LIN {X 0,Y 215.82,Z 913.097,A -85,B 0,C 180,E1 -20872.515,E2 -20872.515} C_VEL
LIN {X 0,Y 216.732,Z 913.858,A -85,B 0,C 180,E1 -20874.417,E2 -20874.417} C_VEL
LIN {X 0,Y 218.187,Z 914.153,A -85,B 0,C 180,E1 -20876.945,E2 -20876.945} C_VEL
LIN {X 0,Y 220.423,Z 913.484,A -85,B 0,C 180,E1 -20880,E2 -20880} C_VEL
LIN {X 0,Y 223.697,Z 911.017,A -85,B 0,C 180,E1 -20883.602,E2 -20883.602} C_VEL
LIN {X 0,Y 226.039,Z 908.76,A -85,B 0,C 180,E1 -20885.743,E2 -20885.743} C_VEL
LIN {X 0,Y 228.842,Z 905.544,A -85,B 0,C 180,E1 -20887.943,E2 -20887.943} C_VEL
LIN {X 0,Y 232.45,Z 900.63,A -85,B 0,C 180,E1 -20890.451,E2 -20890.451} C_VEL
LIN {X 0,Y 236.309,Z 894.485,A -85,B 0,C 180,E1 -20892.888,E2 -20892.888} C_VEL
LIN {X 0,Y 240.084,Z 887.75,A -85,B 0,C 180,E1 -20894.973,E2 -20894.973} C_VEL
LIN {X 0,Y 243.557,Z 880.667,A -85,B 0,C 180,E1 -20896.771,E2 -20896.771} C_VEL
LIN {X 0,Y 246.66,Z 873.613,A -85,B 0,C 180,E1 -20898.265,E2 -20898.265} C_VEL
LIN {X 0,Y 249.838,Z 865.279,A -85,B 0,C 180,E1 -20899.728,E2 -20899.728} C_VEL
LIN {X 0,Y 252.697,Z 856.675,A -85,B 0,C 180,E1 -20900.982,E2 -20900.982} C_VEL
LIN {X 0,Y 255.577,Z 846.343,A -85,B 0,C 180,E1 -20902.216,E2 -20902.216} C_VEL
LIN {X 0,Y 257.749,Z 836.491,A -85,B 0,C 180,E1 -20903.183,E2 -20903.183} C_VEL
LIN {X 0,Y 258.881,Z 830.775,A -85,B 0,C 180,E1 -20903.651,E2 -20903.651} C_VEL
LIN {X 0,Y 259.433,Z 825.363,A -85,B 0,C 180,E1 -20904.174,E2 -20904.174} C_VEL
LIN {X 0,Y 259.323,Z 808.224,A -85,B 0,C 180,E1 -20906.374,E2 -20906.374} C_VEL
LIN {X 0,Y 259.902,Z 802.661,A -85,B 0,C 180,E1 -20906.763,E2 -20906.763} C_VEL
LIN {X 0,Y 261.287,Z 793.546,A -85,B 0,C 180,E1 -20907.21,E2 -20907.21} C_VEL
LIN {X 0,Y 259.496,Z 789.462,A -85,B 0,C 180,E1 -20909.048,E2 -20909.048} C_VEL
LIN {X 0,Y 258.611,Z 787.722,A -85,B 0,C 180,E1 -20910.062,E2 -20910.062} C_VEL
LIN {X 0,Y 257.462,Z 785.023,A -85,B 0,C 180,E1 -20911.841,E2 -20911.841} C_VEL
LIN {X 0,Y 256.142,Z 782.443,A -85,B 0,C 180,E1 -20915.183,E2 -20915.183} C_VEL
LIN {X 0,Y 255.755,Z 782.963,A -85,B 0,C 180,E1 -20917.889,E2 -20917.889} C_VEL
LIN {X 0,Y 256.35,Z 784.832,A -85,B 0,C 180,E1 -20920.768,E2 -20920.768} C_VEL
LIN {X 0,Y 257.554,Z 788.257,A -85,B 0,C 180,E1 -20923.294,E2 -20923.294} C_VEL
LIN {X 0,Y 258.154,Z 798.129,A -85,B 0,C 180,E1 -20925.703,E2 -20925.703} C_VEL
LIN {X 0,Y 256.979,Z 813.634,A -85,B 0,C 180,E1 -20927.292,E2 -20927.292} C_VEL
LIN {X 0,Y 255.567,Z 830.787,A -85,B 0,C 180,E1 -20928.783,E2 -20928.783} C_VEL
LIN {X 0,Y 253.729,Z 848.64,A -85,B 0,C 180,E1 -20929.988,E2 -20929.988} C_VEL
LIN {X 0,Y 251.045,Z 862.414,A -85,B 0,C 180,E1 -20930.697,E2 -20930.697} C_VEL
LIN {X 0,Y 247.953,Z 874.211,A -85,B 0,C 180,E1 -20931.42,E2 -20931.42} C_VEL
LIN {X 0,Y 244.407,Z 885.491,A -85,B 0,C 180,E1 -20932.332,E2 -20932.332} C_VEL
LIN {X 0,Y 240.95,Z 894.919,A -85,B 0,C 180,E1 -20933.275,E2 -20933.275} C_VEL
LIN {X 0,Y 236.566,Z 905.538,A -85,B 0,C 180,E1 -20934.595,E2 -20934.595} C_VEL
LIN {X 0,Y 232.488,Z 914.575,A -85,B 0,C 180,E1 -20935.993,E2 -20935.993} C_VEL
LIN {X 0,Y 228.672,Z 922.392,A -85,B 0,C 180,E1 -20937.46,E2 -20937.46} C_VEL
LIN {X 0,Y 224.196,Z 930.838,A -85,B 0,C 180,E1 -20939.373,E2 -20939.373} C_VEL
LIN {X 0,Y 220.295,Z 938.075,A -85,B 0,C 180,E1 -20941.407,E2 -20941.407} C_VEL
LIN {X 0,Y 216.754,Z 944.309,A -85,B 0,C 180,E1 -20943.521,E2 -20943.521} C_VEL
LIN {X 0,Y 213.717,Z 949.729,A -85,B 0,C 180,E1 -20945.726,E2 -20945.726} C_VEL
LIN {X 0,Y 210.73,Z 955.112,A -85,B 0,C 180,E1 -20948.475,E2 -20948.475} C_VEL
LIN {X 0,Y 208.341,Z 959.496,A -85,B 0,C 180,E1 -20951.306,E2 -20951.306} C_VEL
LIN {X 0,Y 206.818,Z 962.938,A -85,B 0,C 180,E1 -20954.223,E2 -20954.223} C_VEL
LIN {X 0,Y 205.688,Z 966.163,A -85,B 0,C 180,E1 -20958.167,E2 -20958.167} C_VEL
LIN {X 0,Y 205.748,Z 967.832,A -85,B 0,C 180,E1 -20961.564,E2 -20961.564} C_VEL
LIN {X 0,Y 205.939,Z 970.43,A -85,B 0,C 180,E1 -20964.121,E2 -20964.121} C_VEL
LIN {X 0,Y 206.207,Z 971.913,A -85,B 0,C 180,E1 -20966.089,E2 -20966.089} C_VEL
LIN {X 0,Y 206.454,Z 972.92,A -85,B 0,C 180,E1 -20968.046,E2 -20968.046} C_VEL
LIN {X 0,Y 206.718,Z 973.5,A -85,B 0,C 180,E1 -20969.997,E2 -20969.997} C_VEL
LIN {X 0,Y 206.4,Z 973.571,A -85,B 0,C 180,E1 -20971.948,E2 -20971.948} C_VEL
LIN {X 0,Y 206.129,Z 973.197,A -85,B 0,C 180,E1 -20973.907,E2 -20973.907} C_VEL
LIN {X 0,Y 205.527,Z 971.148,A -85,B 0,C 180,E1 -20977.859,E2 -20977.859} C_VEL
LIN {X 0,Y 205.533,Z 968.537,A -85,B 0,C 180,E1 -20980.837,E2 -20980.837} C_VEL
LIN {X 0,Y 206.046,Z 964.96,A -85,B 0,C 180,E1 -20983.81,E2 -20983.81} C_VEL
LIN {X 0,Y 207.188,Z 960.35,A -85,B 0,C 180,E1 -20986.755,E2 -20986.755} C_VEL
LIN {X 0,Y 208.926,Z 954.588,A -85,B 0,C 180,E1 -20989.654,E2 -20989.654} C_VEL
LIN {X 0,Y 211.427,Z 947.534,A -85,B 0,C 180,E1 -20992.471,E2 -20992.471} C_VEL
LIN {X 0,Y 214.497,Z 938.894,A -85,B 0,C 180,E1 -20995.207,E2 -20995.207} C_VEL
LIN {X 0,Y 217.552,Z 930.1,A -85,B 0,C 180,E1 -20997.406,E2 -20997.406} C_VEL
LIN {X 0,Y 221.071,Z 919.363,A -85,B 0,C 180,E1 -20999.518,E2 -20999.518} C_VEL
LIN {X 0,Y 224.586,Z 907.346,A -85,B 0,C 180,E1 -21001.345,E2 -21001.345} C_VEL
LIN {X 0,Y 227.546,Z 895.307,A -85,B 0,C 180,E1 -21002.715,E2 -21002.715} C_VEL
LIN {X 0,Y 229.807,Z 883.048,A -85,B 0,C 180,E1 -21003.778,E2 -21003.778} C_VEL
LIN {X 0,Y 231.633,Z 869.859,A -85,B 0,C 180,E1 -21004.57,E2 -21004.57} C_VEL
LIN {X 0,Y 232.714,Z 855.087,A -85,B 0,C 180,E1 -21005.118,E2 -21005.118} C_VEL
LIN {X 0,Y 233.372,Z 840.252,A -85,B 0,C 180,E1 -21005.6,E2 -21005.6} C_VEL
LIN {X 0,Y 232.16,Z 817.156,A -85,B 0,C 180,E1 -21006.833,E2 -21006.833} C_VEL
LIN {X 0,Y 230.572,Z 796.33,A -85,B 0,C 180,E1 -21008.093,E2 -21008.093} C_VEL
LIN {X 0,Y 228.613,Z 780.544,A -85,B 0,C 180,E1 -21009.258,E2 -21009.258} C_VEL
LIN {X 0,Y 224.716,Z 771.185,A -85,B 0,C 180,E1 -21010.671,E2 -21010.671} C_VEL
LIN {X 0,Y 220.27,Z 761.8,A -85,B 0,C 180,E1 -21012.341,E2 -21012.341} C_VEL
LIN {X 0,Y 216.362,Z 754.458,A -85,B 0,C 180,E1 -21013.9,E2 -21013.9} C_VEL
LIN {X 0,Y 213.79,Z 749.36,A -85,B 0,C 180,E1 -21015.11,E2 -21015.11} C_VEL
LIN {X 0,Y 211.962,Z 742.772,A -85,B 0,C 180,E1 -21018.461,E2 -21018.461} C_VEL
LIN {X 0,Y 209.608,Z 735.268,A -85,B 0,C 180,E1 -21022.877,E2 -21022.877} C_VEL
LIN {X 0,Y 207.43,Z 729.065,A -85,B 0,C 180,E1 -21027.173,E2 -21027.173} C_VEL
LIN {X 0,Y 206.745,Z 726.767,A -85,B 0,C 180,E1 -21029.101,E2 -21029.101} C_VEL
LIN {X 0,Y 206.723,Z 726.734,A -85,B 0,C 180,E1 -21033.771,E2 -21033.771} C_VEL
LIN {X 0,Y 206.747,Z 726.723,A -85,B 0,C 180,E1 -21038.042,E2 -21038.042} C_VEL
LIN {X 0,Y 206.866,Z 726.706,A -85,B 0,C 180,E1 -21042.196,E2 -21042.196} C_VEL
LIN {X 0,Y 206.885,Z 726.703,A -85,B 0,C 180,E1 -21046.244,E2 -21046.244} C_VEL
LIN {X 0,Y 207.088,Z 726.677,A -85,B 0,C 180,E1 -21050.231,E2 -21050.231} C_VEL
LIN {X 0,Y 207.055,Z 726.689,A -85,B 0,C 180,E1 -21054.156,E2 -21054.156} C_VEL
LIN {X 0,Y 207.371,Z 726.655,A -85,B 0,C 180,E1 -21058.058,E2 -21058.058} C_VEL
LIN {X 0,Y 207.504,Z 726.623,A -85,B 0,C 180,E1 -21060,E2 -21060} C_VEL
LIN {X 0,Y 207.371,Z 726.65,A -85,B 0,C 180,E1 -21061.943,E2 -21061.943} C_VEL
LIN {X 0,Y 207.157,Z 726.672,A -85,B 0,C 180,E1 -21067.8,E2 -21067.8} C_VEL
LIN {X 0,Y 206.933,Z 726.7,A -85,B 0,C 180,E1 -21071.758,E2 -21071.758} C_VEL
LIN {X 0,Y 206.906,Z 726.717,A -85,B 0,C 180,E1 -21077.291,E2 -21077.291} C_VEL
LIN {X 0,Y 206.927,Z 727.223,A -85,B 0,C 180,E1 -21078.182,E2 -21078.182} C_VEL
LIN {X 0,Y 207.868,Z 729.668,A -85,B 0,C 180,E1 -21078.896,E2 -21078.896} C_VEL
LIN {X 0,Y 209.947,Z 731.814,A -85,B 0,C 180,E1 -21079.812,E2 -21079.812} C_VEL
LIN {X 0,Y 210.664,Z 732.614,A -85,B 0,C 180,E1 -21080.123,E2 -21080.123} C_VEL
LIN {X 0,Y 212.757,Z 735.862,A -85,B 0,C 180,E1 -21081.054,E2 -21081.054} C_VEL
LIN {X 0,Y 214.374,Z 737.753,A -85,B 0,C 180,E1 -21081.704,E2 -21081.704} C_VEL
LIN {X 0,Y 218.102,Z 743.058,A -85,B 0,C 180,E1 -21083.187,E2 -21083.187} C_VEL
LIN {X 0,Y 221.441,Z 747.9,A -85,B 0,C 180,E1 -21084.428,E2 -21084.428} C_VEL
LIN {X 0,Y 227.298,Z 757.078,A -85,B 0,C 180,E1 -21086.467,E2 -21086.467} C_VEL
LIN {X 0,Y 234.437,Z 769.956,A -85,B 0,C 180,E1 -21088.764,E2 -21088.764} C_VEL
LIN {X 0,Y 236.607,Z 774.439,A -85,B 0,C 180,E1 -21089.441,E2 -21089.441} C_VEL
LIN {X 0,Y 235.209,Z 812.585,A -85,B 0,C 180,E1 -21090.792,E2 -21090.792} C_VEL
LIN {X 0,Y 234.483,Z 825.574,A -85,B 0,C 180,E1 -21091.539,E2 -21091.539} C_VEL
LIN {X 0,Y 233.062,Z 838.159,A -85,B 0,C 180,E1 -21092.588,E2 -21092.588} C_VEL
LIN {X 0,Y 231.265,Z 849.427,A -85,B 0,C 180,E1 -21093.845,E2 -21093.845} C_VEL
LIN {X 0,Y 229.188,Z 859.482,A -85,B 0,C 180,E1 -21095.269,E2 -21095.269} C_VEL
LIN {X 0,Y 226.691,Z 869.468,A -85,B 0,C 180,E1 -21097.035,E2 -21097.035} C_VEL
LIN {X 0,Y 223.982,Z 878.589,A -85,B 0,C 180,E1 -21099.054,E2 -21099.054} C_VEL
LIN {X 0,Y 221.064,Z 887.18,A -85,B 0,C 180,E1 -21101.439,E2 -21101.439} C_VEL
LIN {X 0,Y 218.03,Z 895.011,A -85,B 0,C 180,E1 -21104.18,E2 -21104.18} C_VEL
LIN {X 0,Y 215.643,Z 900.847,A -85,B 0,C 180,E1 -21106.815,E2 -21106.815} C_VEL
LIN {X 0,Y 213.002,Z 906.39,A -85,B 0,C 180,E1 -21110.087,E2 -21110.087} C_VEL
LIN {X 0,Y 211.04,Z 910.178,A -85,B 0,C 180,E1 -21113.175,E2 -21113.175} C_VEL
LIN {X 0,Y 209.998,Z 912.106,A -85,B 0,C 180,E1 -21115.328,E2 -21115.328} C_VEL
LIN {X 0,Y 209.141,Z 913.446,A -85,B 0,C 180,E1 -21117.479,E2 -21117.479} C_VEL
LIN {X 0,Y 208.448,Z 914.316,A -85,B 0,C 180,E1 -21119.623,E2 -21119.623} C_VEL
LIN {X 0,Y 207.976,Z 914.685,A -85,B 0,C 180,E1 -21121.768,E2 -21121.768} C_VEL
LIN {X 0,Y 207.701,Z 914.563,A -85,B 0,C 180,E1 -21123.907,E2 -21123.907} C_VEL
LIN {X 0,Y 207.586,Z 913.993,A -85,B 0,C 180,E1 -21126.081,E2 -21126.081} C_VEL
LIN {X 0,Y 207.696,Z 912.944,A -85,B 0,C 180,E1 -21128.151,E2 -21128.151} C_VEL
LIN {X 0,Y 208.071,Z 910.751,A -85,B 0,C 180,E1 -21131.043,E2 -21131.043} C_VEL
LIN {X 0,Y 209.058,Z 906.954,A -85,B 0,C 180,E1 -21134.402,E2 -21134.402} C_VEL
LIN {X 0,Y 210.273,Z 902.255,A -85,B 0,C 180,E1 -21137.455,E2 -21137.455} C_VEL
LIN {X 0,Y 211.895,Z 896.255,A -85,B 0,C 180,E1 -21140.457,E2 -21140.457} C_VEL
LIN {X 0,Y 213.803,Z 888.74,A -85,B 0,C 180,E1 -21143.396,E2 -21143.396} C_VEL
LIN {X 0,Y 216.063,Z 879.378,A -85,B 0,C 180,E1 -21146.273,E2 -21146.273} C_VEL
LIN {X 0,Y 218.269,Z 869.484,A -85,B 0,C 180,E1 -21148.663,E2 -21148.663} C_VEL
LIN {X 0,Y 220.257,Z 858.973,A -85,B 0,C 180,E1 -21150.688,E2 -21150.688} C_VEL
LIN {X 0,Y 222.265,Z 847.005,A -85,B 0,C 180,E1 -21152.495,E2 -21152.495} C_VEL
LIN {X 0,Y 223.878,Z 834.316,A -85,B 0,C 180,E1 -21153.94,E2 -21153.94} C_VEL
LIN {X 0,Y 224.921,Z 821.294,A -85,B 0,C 180,E1 -21155.044,E2 -21155.044} C_VEL
LIN {X 0,Y 225.492,Z 807.746,A -85,B 0,C 180,E1 -21155.793,E2 -21155.793} C_VEL
LIN {X 0,Y 226.498,Z 770.265,A -85,B 0,C 180,E1 -21157.076,E2 -21157.076} C_VEL
LIN {X 0,Y 226.553,Z 765.8,A -85,B 0,C 180,E1 -21157.236,E2 -21157.236} C_VEL
LIN {X 0,Y 222.198,Z 756.35,A -85,B 0,C 180,E1 -21158.222,E2 -21158.222} C_VEL
LIN {X 0,Y 213.824,Z 739.599,A -85,B 0,C 180,E1 -21160.191,E2 -21160.191} C_VEL
LIN {X 0,Y 208.363,Z 730.146,A -85,B 0,C 180,E1 -21161.514,E2 -21161.514} C_VEL
LIN {X 0,Y 207.034,Z 727.418,A -85,B 0,C 180,E1 -21161.941,E2 -21161.941} C_VEL
LIN {X 0,Y 206.907,Z 726.757,A -85,B 0,C 180,E1 -21162.384,E2 -21162.384} C_VEL
LIN {X 0,Y 206.814,Z 726.719,A -85,B 0,C 180,E1 -21167.915,E2 -21167.915} C_VEL
LIN {X 0,Y 206.732,Z 726.734,A -85,B 0,C 180,E1 -21173.38,E2 -21173.38} C_VEL
LIN {X 0,Y 206.685,Z 726.721,A -85,B 0,C 180,E1 -21178.431,E2 -21178.431} C_VEL
LIN {X 0,Y 206.699,Z 726.709,A -85,B 0,C 180,E1 -21182.961,E2 -21182.961} C_VEL
LIN {X 0,Y 206.707,Z 726.693,A -85,B 0,C 180,E1 -21185.313,E2 -21185.313} C_VEL
LIN {X 0,Y 206.654,Z 726.743,A -85,B 0,C 180,E1 -21190.256,E2 -21190.256} C_VEL
LIN {X 0,Y 206.637,Z 726.746,A -85,B 0,C 180,E1 -21194.418,E2 -21194.418} C_VEL
LIN {X 0,Y 206.706,Z 726.866,A -85,B 0,C 180,E1 -21197.499,E2 -21197.499} C_VEL
LIN {X 0,Y 206.93,Z 727.899,A -85,B 0,C 180,E1 -21197.85,E2 -21197.85} C_VEL
LIN {X 0,Y 216.887,Z 756.802,A -85,B 0,C 180,E1 -21200.104,E2 -21200.104} C_VEL
LIN {X 0,Y 214.902,Z 807.381,A -85,B 0,C 180,E1 -21202.586,E2 -21202.586} C_VEL
LIN {X 0,Y 214.443,Z 818.809,A -85,B 0,C 180,E1 -21203.411,E2 -21203.411} C_VEL
LIN {X 0,Y 213.661,Z 829.523,A -85,B 0,C 180,E1 -21204.421,E2 -21204.421} C_VEL
LIN {X 0,Y 212.813,Z 839.899,A -85,B 0,C 180,E1 -21205.655,E2 -21205.655} C_VEL
LIN {X 0,Y 211.854,Z 849.82,A -85,B 0,C 180,E1 -21207.096,E2 -21207.096} C_VEL
LIN {X 0,Y 210.982,Z 858.654,A -85,B 0,C 180,E1 -21208.635,E2 -21208.635} C_VEL
LIN {X 0,Y 210.053,Z 867.479,A -85,B 0,C 180,E1 -21210.454,E2 -21210.454} C_VEL
LIN {X 0,Y 209.101,Z 875.776,A -85,B 0,C 180,E1 -21212.474,E2 -21212.474} C_VEL
LIN {X 0,Y 208.331,Z 882.894,A -85,B 0,C 180,E1 -21214.521,E2 -21214.521} C_VEL
LIN {X 0,Y 207.784,Z 889.046,A -85,B 0,C 180,E1 -21216.582,E2 -21216.582} C_VEL
LIN {X 0,Y 207.253,Z 895.478,A -85,B 0,C 180,E1 -21219.141,E2 -21219.141} C_VEL
LIN {X 0,Y 206.951,Z 901.32,A -85,B 0,C 180,E1 -21221.973,E2 -21221.973} C_VEL
LIN {X 0,Y 206.941,Z 905.217,A -85,B 0,C 180,E1 -21224.235,E2 -21224.235} C_VEL
LIN {X 0,Y 207.252,Z 909.316,A -85,B 0,C 180,E1 -21227.266,E2 -21227.266} C_VEL
LIN {X 0,Y 207.969,Z 912.307,A -85,B 0,C 180,E1 -21230.272,E2 -21230.272} C_VEL
LIN {X 0,Y 208.666,Z 913.803,A -85,B 0,C 180,E1 -21232.257,E2 -21232.257} C_VEL
LIN {X 0,Y 209.561,Z 914.771,A -85,B 0,C 180,E1 -21234.225,E2 -21234.225} C_VEL
LIN {X 0,Y 211.138,Z 915.431,A -85,B 0,C 180,E1 -21237,E2 -21237} C_VEL
LIN {X 0,Y 213.32,Z 915.036,A -85,B 0,C 180,E1 -21240,E2 -21240} C_VEL
LIN {X 0,Y 216.762,Z 913.224,A -85,B 0,C 180,E1 -21243.718,E2 -21243.718} C_VEL
LIN {X 0,Y 218.997,Z 911.285,A -85,B 0,C 180,E1 -21245.798,E2 -21245.798} C_VEL
LIN {X 0,Y 223.257,Z 907.003,A -85,B 0,C 180,E1 -21249.056,E2 -21249.056} C_VEL
LIN {X 0,Y 227.125,Z 902.208,A -85,B 0,C 180,E1 -21251.603,E2 -21251.603} C_VEL
LIN {X 0,Y 231.238,Z 896.108,A -85,B 0,C 180,E1 -21254.072,E2 -21254.072} C_VEL
LIN {X 0,Y 234.902,Z 890.204,A -85,B 0,C 180,E1 -21255.978,E2 -21255.978} C_VEL
LIN {X 0,Y 238.986,Z 882.509,A -85,B 0,C 180,E1 -21257.986,E2 -21257.986} C_VEL
LIN {X 0,Y 242.256,Z 875.569,A -85,B 0,C 180,E1 -21259.489,E2 -21259.489} C_VEL
LIN {X 0,Y 246.064,Z 866.289,A -85,B 0,C 180,E1 -21261.136,E2 -21261.136} C_VEL
LIN {X 0,Y 249.093,Z 857.65,A -85,B 0,C 180,E1 -21262.389,E2 -21262.389} C_VEL
LIN {X 0,Y 252.156,Z 847.308,A -85,B 0,C 180,E1 -21263.619,E2 -21263.619} C_VEL
LIN {X 0,Y 254.264,Z 838.512,A -85,B 0,C 180,E1 -21264.495,E2 -21264.495} C_VEL
LIN {X 0,Y 256.275,Z 827.99,A -85,B 0,C 180,E1 -21265.318,E2 -21265.318} C_VEL
LIN {X 0,Y 259.053,Z 808.51,A -85,B 0,C 180,E1 -21266.461,E2 -21266.461} C_VEL
LIN {X 0,Y 259.902,Z 802.661,A -85,B 0,C 180,E1 -21266.763,E2 -21266.763} C_VEL
LIN {X 0,Y 260.053,Z 800.423,A -85,B 0,C 180,E1 -21266.989,E2 -21266.989} C_VEL
LIN {X 0,Y 259.657,Z 797.879,A -85,B 0,C 180,E1 -21267.614,E2 -21267.614} C_VEL
LIN {X 0,Y 258.867,Z 796.265,A -85,B 0,C 180,E1 -21268.397,E2 -21268.397} C_VEL
LIN {X 0,Y 256.343,Z 793.547,A -85,B 0,C 180,E1 -21270.964,E2 -21270.964} C_VEL
LIN {X 0,Y 255.705,Z 791.806,A -85,B 0,C 180,E1 -21272.085,E2 -21272.085} C_VEL
LIN {X 0,Y 254.611,Z 789.403,A -85,B 0,C 180,E1 -21275.106,E2 -21275.106} C_VEL
LIN {X 0,Y 254.203,Z 789.877,A -85,B 0,C 180,E1 -21277.762,E2 -21277.762} C_VEL
LIN {X 0,Y 254.623,Z 791.518,A -85,B 0,C 180,E1 -21280.389,E2 -21280.389} C_VEL
LIN {X 0,Y 255.484,Z 794.383,A -85,B 0,C 180,E1 -21282.575,E2 -21282.575} C_VEL
LIN {X 0,Y 255.639,Z 802.165,A -85,B 0,C 180,E1 -21284.479,E2 -21284.479} C_VEL
LIN {X 0,Y 254.273,Z 816.273,A -85,B 0,C 180,E1 -21285.941,E2 -21285.941} C_VEL
LIN {X 0,Y 252.682,Z 832.423,A -85,B 0,C 180,E1 -21287.367,E2 -21287.367} C_VEL
LIN {X 0,Y 250.462,Z 850.054,A -85,B 0,C 180,E1 -21288.591,E2 -21288.591} C_VEL
LIN {X 0,Y 247.701,Z 862.896,A -85,B 0,C 180,E1 -21289.261,E2 -21289.261} C_VEL
LIN {X 0,Y 244.486,Z 874.147,A -85,B 0,C 180,E1 -21289.967,E2 -21289.967} C_VEL
LIN {X 0,Y 240.797,Z 885.027,A -85,B 0,C 180,E1 -21290.862,E2 -21290.862} C_VEL
LIN {X 0,Y 237.153,Z 894.248,A -85,B 0,C 180,E1 -21291.781,E2 -21291.781} C_VEL
LIN {X 0,Y 233.147,Z 903.487,A -85,B 0,C 180,E1 -21292.921,E2 -21292.921} C_VEL
LIN {X 0,Y 228.862,Z 912.503,A -85,B 0,C 180,E1 -21294.303,E2 -21294.303} C_VEL
LIN {X 0,Y 224.727,Z 920.371,A -85,B 0,C 180,E1 -21295.739,E2 -21295.739} C_VEL
LIN {X 0,Y 219.967,Z 928.861,A -85,B 0,C 180,E1 -21297.642,E2 -21297.642} C_VEL
LIN {X 0,Y 215.701,Z 936.111,A -85,B 0,C 180,E1 -21299.664,E2 -21299.664} C_VEL
LIN {X 0,Y 211.116,Z 943.51,A -85,B 0,C 180,E1 -21302.218,E2 -21302.218} C_VEL
LIN {X 0,Y 207.265,Z 949.679,A -85,B 0,C 180,E1 -21304.919,E2 -21304.919} C_VEL
LIN {X 0,Y 204.108,Z 954.791,A -85,B 0,C 180,E1 -21307.74,E2 -21307.74} C_VEL
LIN {X 0,Y 201.875,Z 958.451,A -85,B 0,C 180,E1 -21310.237,E2 -21310.237} C_VEL
LIN {X 0,Y 199.935,Z 962.196,A -85,B 0,C 180,E1 -21313.665,E2 -21313.665} C_VEL
LIN {X 0,Y 198.696,Z 965.18,A -85,B 0,C 180,E1 -21317.744,E2 -21317.744} C_VEL
LIN {X 0,Y 198.702,Z 966.744,A -85,B 0,C 180,E1 -21321.351,E2 -21321.351} C_VEL
LIN {X 0,Y 198.873,Z 969.272,A -85,B 0,C 180,E1 -21323.911,E2 -21323.911} C_VEL
LIN {X 0,Y 199.149,Z 970.809,A -85,B 0,C 180,E1 -21325.95,E2 -21325.95} C_VEL
LIN {X 0,Y 199.401,Z 971.844,A -85,B 0,C 180,E1 -21327.977,E2 -21327.977} C_VEL
LIN {X 0,Y 199.682,Z 972.45,A -85,B 0,C 180,E1 -21329.997,E2 -21329.997} C_VEL
LIN {X 0,Y 199.347,Z 972.54,A -85,B 0,C 180,E1 -21332.017,E2 -21332.017} C_VEL
LIN {X 0,Y 199.041,Z 972.204,A -85,B 0,C 180,E1 -21334.046,E2 -21334.046} C_VEL
LIN {X 0,Y 198.437,Z 970.195,A -85,B 0,C 180,E1 -21338.141,E2 -21338.141} C_VEL
LIN {X 0,Y 198.498,Z 967.63,A -85,B 0,C 180,E1 -21341.226,E2 -21341.226} C_VEL
LIN {X 0,Y 199.467,Z 962.735,A -85,B 0,C 180,E1 -21345.319,E2 -21345.319} C_VEL
LIN {X 0,Y 201.097,Z 956.812,A -85,B 0,C 180,E1 -21348.887,E2 -21348.887} C_VEL
LIN {X 0,Y 203.918,Z 949.404,A -85,B 0,C 180,E1 -21352.275,E2 -21352.275} C_VEL
LIN {X 0,Y 206.892,Z 941.419,A -85,B 0,C 180,E1 -21355.123,E2 -21355.123} C_VEL
LIN {X 0,Y 210.573,Z 931.527,A -85,B 0,C 180,E1 -21357.853,E2 -21357.853} C_VEL
LIN {X 0,Y 214.133,Z 921.422,A -85,B 0,C 180,E1 -21360.031,E2 -21360.031} C_VEL
LIN {X 0,Y 217.721,Z 910.154,A -85,B 0,C 180,E1 -21361.906,E2 -21361.906} C_VEL
LIN {X 0,Y 221.189,Z 897.469,A -85,B 0,C 180,E1 -21363.505,E2 -21363.505} C_VEL
LIN {X 0,Y 223.631,Z 885.569,A -85,B 0,C 180,E1 -21364.658,E2 -21364.658} C_VEL
LIN {X 0,Y 225.689,Z 872.92,A -85,B 0,C 180,E1 -21365.507,E2 -21365.507} C_VEL
LIN {X 0,Y 227.003,Z 859.434,A -85,B 0,C 180,E1 -21366.113,E2 -21366.113} C_VEL
LIN {X 0,Y 227.942,Z 841.187,A -85,B 0,C 180,E1 -21366.713,E2 -21366.713} C_VEL
LIN {X 0,Y 226.856,Z 818.463,A -85,B 0,C 180,E1 -21367.96,E2 -21367.96} C_VEL
LIN {X 0,Y 225.377,Z 797.977,A -85,B 0,C 180,E1 -21369.241,E2 -21369.241} C_VEL
LIN {X 0,Y 223.666,Z 783.414,A -85,B 0,C 180,E1 -21370.361,E2 -21370.361} C_VEL
LIN {X 0,Y 218.955,Z 772.046,A -85,B 0,C 180,E1 -21372.199,E2 -21372.199} C_VEL
LIN {X 0,Y 215.336,Z 764.793,A -85,B 0,C 180,E1 -21373.657,E2 -21373.657} C_VEL
LIN {X 0,Y 212.406,Z 759.065,A -85,B 0,C 180,E1 -21374.912,E2 -21374.912} C_VEL
LIN {X 0,Y 209.379,Z 753.488,A -85,B 0,C 180,E1 -21376.263,E2 -21376.263} C_VEL
LIN {X 0,Y 206.131,Z 747.484,A -85,B 0,C 180,E1 -21377.92,E2 -21377.92} C_VEL
LIN {X 0,Y 204.145,Z 740.919,A -85,B 0,C 180,E1 -21381.708,E2 -21381.708} C_VEL
LIN {X 0,Y 202.538,Z 735.846,A -85,B 0,C 180,E1 -21385.072,E2 -21385.072} C_VEL
LIN {X 0,Y 200.499,Z 730.176,A -85,B 0,C 180,E1 -21389.452,E2 -21389.452} C_VEL
LIN {X 0,Y 199.705,Z 727.647,A -85,B 0,C 180,E1 -21391.81,E2 -21391.81} C_VEL
LIN {X 0,Y 199.728,Z 727.605,A -85,B 0,C 180,E1 -21397.228,E2 -21397.228} C_VEL
LIN {X 0,Y 199.827,Z 727.585,A -85,B 0,C 180,E1 -21401.721,E2 -21401.721} C_VEL
LIN {X 0,Y 199.825,Z 727.585,A -85,B 0,C 180,E1 -21405.748,E2 -21405.748} C_VEL
LIN {X 0,Y 200.011,Z 727.562,A -85,B 0,C 180,E1 -21409.881,E2 -21409.881} C_VEL
LIN {X 0,Y 200.017,Z 727.568,A -85,B 0,C 180,E1 -21413.949,E2 -21413.949} C_VEL
LIN {X 0,Y 200.311,Z 727.534,A -85,B 0,C 180,E1 -21417.99,E2 -21417.99} C_VEL
LIN {X 0,Y 200.469,Z 727.499,A -85,B 0,C 180,E1 -21420,E2 -21420} C_VEL
LIN {X 0,Y 200.02,Z 727.557,A -85,B 0,C 180,E1 -21424.03,E2 -21424.03} C_VEL
LIN {X 0,Y 200.101,Z 727.549,A -85,B 0,C 180,E1 -21428.077,E2 -21428.077} C_VEL
LIN {X 0,Y 199.876,Z 727.577,A -85,B 0,C 180,E1 -21432.18,E2 -21432.18} C_VEL
LIN {X 0,Y 199.838,Z 727.852,A -85,B 0,C 180,E1 -21434.968,E2 -21434.968} C_VEL
LIN {X 0,Y 200.137,Z 729.01,A -85,B 0,C 180,E1 -21435.531,E2 -21435.531} C_VEL
LIN {X 0,Y 201.853,Z 731.746,A -85,B 0,C 180,E1 -21436.545,E2 -21436.545} C_VEL
LIN {X 0,Y 203.812,Z 733.309,A -85,B 0,C 180,E1 -21437.502,E2 -21437.502} C_VEL
LIN {X 0,Y 205.68,Z 736.495,A -85,B 0,C 180,E1 -21438.471,E2 -21438.471} C_VEL
LIN {X 0,Y 207.63,Z 738.565,A -85,B 0,C 180,E1 -21439.361,E2 -21439.361} C_VEL
LIN {X 0,Y 210.238,Z 742.272,A -85,B 0,C 180,E1 -21440.549,E2 -21440.549} C_VEL
LIN {X 0,Y 214.782,Z 748.678,A -85,B 0,C 180,E1 -21442.446,E2 -21442.446} C_VEL
LIN {X 0,Y 220.896,Z 757.948,A -85,B 0,C 180,E1 -21444.782,E2 -21444.782} C_VEL
LIN {X 0,Y 227.899,Z 770.287,A -85,B 0,C 180,E1 -21447.244,E2 -21447.244} C_VEL
LIN {X 0,Y 231.266,Z 776.959,A -85,B 0,C 180,E1 -21448.349,E2 -21448.349} C_VEL
LIN {X 0,Y 229.758,Z 815.245,A -85,B 0,C 180,E1 -21449.744,E2 -21449.744} C_VEL
LIN {X 0,Y 228.872,Z 828.24,A -85,B 0,C 180,E1 -21450.558,E2 -21450.558} C_VEL
LIN {X 0,Y 227.299,Z 841.139,A -85,B 0,C 180,E1 -21451.711,E2 -21451.711} C_VEL
LIN {X 0,Y 225.278,Z 852.356,A -85,B 0,C 180,E1 -21453.032,E2 -21453.032} C_VEL
LIN {X 0,Y 223.025,Z 862.403,A -85,B 0,C 180,E1 -21454.557,E2 -21454.557} C_VEL
LIN {X 0,Y 219.998,Z 873.231,A -85,B 0,C 180,E1 -21456.623,E2 -21456.623} C_VEL
LIN {X 0,Y 216.873,Z 882.851,A -85,B 0,C 180,E1 -21458.95,E2 -21458.95} C_VEL
LIN {X 0,Y 213.712,Z 891.303,A -85,B 0,C 180,E1 -21461.575,E2 -21461.575} C_VEL
LIN {X 0,Y 210.614,Z 898.65,A -85,B 0,C 180,E1 -21464.488,E2 -21464.488} C_VEL
LIN {X 0,Y 207.945,Z 904.443,A -85,B 0,C 180,E1 -21467.477,E2 -21467.477} C_VEL
LIN {X 0,Y 205.457,Z 909.162,A -85,B 0,C 180,E1 -21470.745,E2 -21470.745} C_VEL
LIN {X 0,Y 203.549,Z 912.514,A -85,B 0,C 180,E1 -21474.062,E2 -21474.062} C_VEL
LIN {X 0,Y 202.507,Z 914.151,A -85,B 0,C 180,E1 -21476.401,E2 -21476.401} C_VEL
LIN {X 0,Y 201.748,Z 915.093,A -85,B 0,C 180,E1 -21478.501,E2 -21478.501} C_VEL
LIN {X 0,Y 201.142,Z 915.651,A -85,B 0,C 180,E1 -21480.871,E2 -21480.871} C_VEL
LIN {X 0,Y 200.776,Z 915.702,A -85,B 0,C 180,E1 -21482.935,E2 -21482.935} C_VEL
LIN {X 0,Y 200.587,Z 915.111,A -85,B 0,C 180,E1 -21485.641,E2 -21485.641} C_VEL
LIN {X 0,Y 200.792,Z 913.049,A -85,B 0,C 180,E1 -21489.515,E2 -21489.515} C_VEL
LIN {X 0,Y 201.459,Z 910.13,A -85,B 0,C 180,E1 -21492.754,E2 -21492.754} C_VEL
LIN {X 0,Y 202.666,Z 905.753,A -85,B 0,C 180,E1 -21496.165,E2 -21496.165} C_VEL
LIN {X 0,Y 204.234,Z 899.86,A -85,B 0,C 180,E1 -21499.595,E2 -21499.595} C_VEL
LIN {X 0,Y 206.131,Z 892.951,A -85,B 0,C 180,E1 -21502.657,E2 -21502.657} C_VEL
LIN {X 0,Y 208.381,Z 884.367,A -85,B 0,C 180,E1 -21505.651,E2 -21505.651} C_VEL
LIN {X 0,Y 210.504,Z 875.598,A -85,B 0,C 180,E1 -21508.09,E2 -21508.09} C_VEL
LIN {X 0,Y 212.81,Z 864.767,A -85,B 0,C 180,E1 -21510.476,E2 -21510.476} C_VEL
LIN {X 0,Y 214.843,Z 854.02,A -85,B 0,C 180,E1 -21512.346,E2 -21512.346} C_VEL
LIN {X 0,Y 216.654,Z 842.192,A -85,B 0,C 180,E1 -21513.955,E2 -21513.955} C_VEL
LIN {X 0,Y 217.957,Z 830.145,A -85,B 0,C 180,E1 -21515.206,E2 -21515.206} C_VEL
LIN {X 0,Y 218.868,Z 817.193,A -85,B 0,C 180,E1 -21516.178,E2 -21516.178} C_VEL
LIN {X 0,Y 219.273,Z 803.768,A -85,B 0,C 180,E1 -21516.813,E2 -21516.813} C_VEL
LIN {X 0,Y 220.337,Z 767.785,A -85,B 0,C 180,E1 -21518.054,E2 -21518.054} C_VEL
LIN {X 0,Y 215.093,Z 756.745,A -85,B 0,C 180,E1 -21519.294,E2 -21519.294} C_VEL
LIN {X 0,Y 208.05,Z 742.583,A -85,B 0,C 180,E1 -21521.041,E2 -21521.041} C_VEL
LIN {X 0,Y 201.128,Z 730.858,A -85,B 0,C 180,E1 -21522.802,E2 -21522.802} C_VEL
LIN {X 0,Y 199.941,Z 728.206,A -85,B 0,C 180,E1 -21523.243,E2 -21523.243} C_VEL
LIN {X 0,Y 199.839,Z 727.622,A -85,B 0,C 180,E1 -21523.787,E2 -21523.787} C_VEL
LIN {X 0,Y 199.729,Z 727.592,A -85,B 0,C 180,E1 -21528.466,E2 -21528.466} C_VEL
LIN {X 0,Y 199.691,Z 727.607,A -85,B 0,C 180,E1 -21533.785,E2 -21533.785} C_VEL
LIN {X 0,Y 199.662,Z 727.594,A -85,B 0,C 180,E1 -21538.358,E2 -21538.358} C_VEL
LIN {X 0,Y 199.671,Z 727.593,A -85,B 0,C 180,E1 -21542.354,E2 -21542.354} C_VEL
LIN {X 0,Y 199.624,Z 727.587,A -85,B 0,C 180,E1 -21546.766,E2 -21546.766} C_VEL
LIN {X 0,Y 199.602,Z 727.621,A -85,B 0,C 180,E1 -21549.333,E2 -21549.333} C_VEL
LIN {X 0,Y 199.573,Z 727.626,A -85,B 0,C 180,E1 -21552.309,E2 -21552.309} C_VEL
LIN {X 0,Y 199.656,Z 727.773,A -85,B 0,C 180,E1 -21557,E2 -21557} C_VEL
LIN {X 0,Y 199.894,Z 728.803,A -85,B 0,C 180,E1 -21557.343,E2 -21557.343} C_VEL
LIN {X 0,Y 209.931,Z 757.972,A -85,B 0,C 180,E1 -21559.705,E2 -21559.705} C_VEL
LIN {X 0,Y 207.924,Z 808.694,A -85,B 0,C 180,E1 -21562.295,E2 -21562.295} C_VEL
LIN {X 0,Y 207.38,Z 820.322,A -85,B 0,C 180,E1 -21563.171,E2 -21563.171} C_VEL
LIN {X 0,Y 206.623,Z 830.996,A -85,B 0,C 180,E1 -21564.224,E2 -21564.224} C_VEL
LIN {X 0,Y 205.783,Z 840.621,A -85,B 0,C 180,E1 -21565.404,E2 -21565.404} C_VEL
LIN {X 0,Y 204.907,Z 849.488,A -85,B 0,C 180,E1 -21566.716,E2 -21566.716} C_VEL
LIN {X 0,Y 203.996,Z 858.496,A -85,B 0,C 180,E1 -21568.305,E2 -21568.305} C_VEL
LIN {X 0,Y 202.994,Z 867.837,A -85,B 0,C 180,E1 -21570.273,E2 -21570.273} C_VEL
LIN {X 0,Y 202.155,Z 874.934,A -85,B 0,C 180,E1 -21572.008,E2 -21572.008} C_VEL
LIN {X 0,Y 201.327,Z 882.363,A -85,B 0,C 180,E1 -21574.128,E2 -21574.128} C_VEL
LIN {X 0,Y 200.611,Z 890.137,A -85,B 0,C 180,E1 -21576.788,E2 -21576.788} C_VEL
LIN {X 0,Y 200.117,Z 896.598,A -85,B 0,C 180,E1 -21579.439,E2 -21579.439} C_VEL
LIN {X 0,Y 199.889,Z 901.286,A -85,B 0,C 180,E1 -21581.687,E2 -21581.687} C_VEL
LIN {X 0,Y 199.886,Z 906.373,A -85,B 0,C 180,E1 -21584.71,E2 -21584.71} C_VEL
LIN {X 0,Y 200.292,Z 910.479,A -85,B 0,C 180,E1 -21587.846,E2 -21587.846} C_VEL
LIN {X 0,Y 200.785,Z 912.672,A -85,B 0,C 180,E1 -21589.92,E2 -21589.92} C_VEL
LIN {X 0,Y 202.367,Z 915.56,A -85,B 0,C 180,E1 -21594.019,E2 -21594.019} C_VEL
LIN {X 0,Y 204.088,Z 916.586,A -85,B 0,C 180,E1 -21597.066,E2 -21597.066} C_VEL
LIN {X 0,Y 206.221,Z 916.598,A -85,B 0,C 180,E1 -21600,E2 -21600} C_VEL
LIN {X 0,Y 207.895,Z 916.158,A -85,B 0,C 180,E1 -21601.937,E2 -21601.937} C_VEL
LIN {X 0,Y 211.979,Z 913.667,A -85,B 0,C 180,E1 -21605.918,E2 -21605.918} C_VEL
LIN {X 0,Y 215.206,Z 910.999,A -85,B 0,C 180,E1 -21608.45,E2 -21608.45} C_VEL
LIN {X 0,Y 219.088,Z 907.025,A -85,B 0,C 180,E1 -21611.097,E2 -21611.097} C_VEL
LIN {X 0,Y 221.9,Z 903.838,A -85,B 0,C 180,E1 -21612.809,E2 -21612.809} C_VEL
LIN {X 0,Y 226.277,Z 897.972,A -85,B 0,C 180,E1 -21615.266,E2 -21615.266} C_VEL
LIN {X 0,Y 231.165,Z 890.364,A -85,B 0,C 180,E1 -21617.699,E2 -21617.699} C_VEL
LIN {X 0,Y 234.563,Z 884.5,A -85,B 0,C 180,E1 -21619.243,E2 -21619.243} C_VEL
LIN {X 0,Y 238.902,Z 875.743,A -85,B 0,C 180,E1 -21621.123,E2 -21621.123} C_VEL
LIN {X 0,Y 242.509,Z 867.458,A -85,B 0,C 180,E1 -21622.581,E2 -21622.581} C_VEL
LIN {X 0,Y 245.756,Z 858.861,A -85,B 0,C 180,E1 -21623.822,E2 -21623.822} C_VEL
LIN {X 0,Y 248.472,Z 850.306,A -85,B 0,C 180,E1 -21624.859,E2 -21624.859} C_VEL
LIN {X 0,Y 251.225,Z 839.769,A -85,B 0,C 180,E1 -21625.919,E2 -21625.919} C_VEL
LIN {X 0,Y 253.435,Z 828.895,A -85,B 0,C 180,E1 -21626.784,E2 -21626.784} C_VEL
LIN {X 0,Y 256.911,Z 806.243,A -85,B 0,C 180,E1 -21628.085,E2 -21628.085} C_VEL
LIN {X 0,Y 258.229,Z 797.995,A -85,B 0,C 180,E1 -21628.514,E2 -21628.514} C_VEL
LIN {X 0,Y 256.753,Z 794.433,A -85,B 0,C 180,E1 -21630.35,E2 -21630.35} C_VEL
LIN {X 0,Y 256.343,Z 793.547,A -85,B 0,C 180,E1 -21630.964,E2 -21630.964} C_VEL
LIN {X 0,Y 255.418,Z 792.685,A -85,B 0,C 180,E1 -21632.257,E2 -21632.257} C_VEL
LIN {X 0,Y 254.453,Z 793.053,A -85,B 0,C 180,E1 -21633.576,E2 -21633.576} C_VEL
LIN {X 0,Y 252.721,Z 796.414,A -85,B 0,C 180,E1 -21637.145,E2 -21637.145} C_VEL
LIN {X 0,Y 252.623,Z 797.023,A -85,B 0,C 180,E1 -21638.058,E2 -21638.058} C_VEL
LIN {X 0,Y 252.978,Z 798.516,A -85,B 0,C 180,E1 -21640.261,E2 -21640.261} C_VEL
LIN {X 0,Y 253.5,Z 800.771,A -85,B 0,C 180,E1 -21641.903,E2 -21641.903} C_VEL
LIN {X 0,Y 253.393,Z 806.34,A -85,B 0,C 180,E1 -21643.248,E2 -21643.248} C_VEL
LIN {X 0,Y 251.686,Z 820.344,A -85,B 0,C 180,E1 -21644.684,E2 -21644.684} C_VEL
LIN {X 0,Y 249.872,Z 835.707,A -85,B 0,C 180,E1 -21646.034,E2 -21646.034} C_VEL
LIN {X 0,Y 247.562,Z 851.28,A -85,B 0,C 180,E1 -21647.119,E2 -21647.119} C_VEL
LIN {X 0,Y 244.552,Z 863.757,A -85,B 0,C 180,E1 -21647.794,E2 -21647.794} C_VEL
LIN {X 0,Y 239.937,Z 878.223,A -85,B 0,C 180,E1 -21648.77,E2 -21648.77} C_VEL
LIN {X 0,Y 234.817,Z 891.062,A -85,B 0,C 180,E1 -21649.945,E2 -21649.945} C_VEL
LIN {X 0,Y 229.942,Z 901.682,A -85,B 0,C 180,E1 -21651.2,E2 -21651.2} C_VEL
LIN {X 0,Y 225.391,Z 910.65,A -85,B 0,C 180,E1 -21652.549,E2 -21652.549} C_VEL
LIN {X 0,Y 221.073,Z 918.543,A -85,B 0,C 180,E1 -21653.973,E2 -21653.973} C_VEL
LIN {X 0,Y 216.005,Z 927.003,A -85,B 0,C 180,E1 -21655.855,E2 -21655.855} C_VEL
LIN {X 0,Y 211.381,Z 934.281,A -85,B 0,C 180,E1 -21657.858,E2 -21657.858} C_VEL
LIN {X 0,Y 206.403,Z 941.694,A -85,B 0,C 180,E1 -21660.411,E2 -21660.411} C_VEL
LIN {X 0,Y 202.123,Z 947.889,A -85,B 0,C 180,E1 -21663.123,E2 -21663.123} C_VEL
LIN {X 0,Y 198.537,Z 953.045,A -85,B 0,C 180,E1 -21665.975,E2 -21665.975} C_VEL
LIN {X 0,Y 195.362,Z 957.609,A -85,B 0,C 180,E1 -21669.281,E2 -21669.281} C_VEL
LIN {X 0,Y 193.074,Z 961.387,A -85,B 0,C 180,E1 -21673.067,E2 -21673.067} C_VEL
LIN {X 0,Y 192.203,Z 963.01,A -85,B 0,C 180,E1 -21675.166,E2 -21675.166} C_VEL
LIN {X 0,Y 191.565,Z 964.959,A -85,B 0,C 180,E1 -21679.427,E2 -21679.427} C_VEL
LIN {X 0,Y 191.645,Z 965.54,A -85,B 0,C 180,E1 -21681.03,E2 -21681.03} C_VEL
LIN {X 0,Y 191.794,Z 968.112,A -85,B 0,C 180,E1 -21683.686,E2 -21683.686} C_VEL
LIN {X 0,Y 192.092,Z 969.693,A -85,B 0,C 180,E1 -21685.801,E2 -21685.801} C_VEL
LIN {X 0,Y 192.346,Z 970.767,A -85,B 0,C 180,E1 -21687.903,E2 -21687.903} C_VEL
LIN {X 0,Y 192.643,Z 971.399,A -85,B 0,C 180,E1 -21689.997,E2 -21689.997} C_VEL
LIN {X 0,Y 192.291,Z 971.508,A -85,B 0,C 180,E1 -21692.091,E2 -21692.091} C_VEL
LIN {X 0,Y 191.955,Z 971.199,A -85,B 0,C 180,E1 -21694.196,E2 -21694.196} C_VEL
LIN {X 0,Y 191.442,Z 969.775,A -85,B 0,C 180,E1 -21697.611,E2 -21697.611} C_VEL
LIN {X 0,Y 191.376,Z 967.676,A -85,B 0,C 180,E1 -21700.577,E2 -21700.577} C_VEL
LIN {X 0,Y 191.855,Z 964.53,A -85,B 0,C 180,E1 -21703.771,E2 -21703.771} C_VEL
LIN {X 0,Y 192.981,Z 960.394,A -85,B 0,C 180,E1 -21706.935,E2 -21706.935} C_VEL
LIN {X 0,Y 195.013,Z 954.418,A -85,B 0,C 180,E1 -21710.446,E2 -21710.446} C_VEL
LIN {X 0,Y 197.803,Z 947.555,A -85,B 0,C 180,E1 -21713.557,E2 -21713.557} C_VEL
LIN {X 0,Y 201.079,Z 939.356,A -85,B 0,C 180,E1 -21716.46,E2 -21716.46} C_VEL
LIN {X 0,Y 205.032,Z 929.297,A -85,B 0,C 180,E1 -21719.235,E2 -21719.235} C_VEL
LIN {X 0,Y 208.853,Z 918.932,A -85,B 0,C 180,E1 -21721.435,E2 -21721.435} C_VEL
LIN {X 0,Y 212.624,Z 907.321,A -85,B 0,C 180,E1 -21723.33,E2 -21723.33} C_VEL
LIN {X 0,Y 215.756,Z 895.994,A -85,B 0,C 180,E1 -21724.749,E2 -21724.749} C_VEL
LIN {X 0,Y 218.49,Z 883.168,A -85,B 0,C 180,E1 -21725.963,E2 -21725.963} C_VEL
LIN {X 0,Y 220.551,Z 870.347,A -85,B 0,C 180,E1 -21726.806,E2 -21726.806} C_VEL
LIN {X 0,Y 221.8,Z 857.406,A -85,B 0,C 180,E1 -21727.37,E2 -21727.37} C_VEL
LIN {X 0,Y 222.571,Z 841.449,A -85,B 0,C 180,E1 -21727.918,E2 -21727.918} C_VEL
LIN {X 0,Y 221.571,Z 818.477,A -85,B 0,C 180,E1 -21729.226,E2 -21729.226} C_VEL
LIN {X 0,Y 220.336,Z 799.64,A -85,B 0,C 180,E1 -21730.45,E2 -21730.45} C_VEL
LIN {X 0,Y 218.946,Z 786.643,A -85,B 0,C 180,E1 -21731.469,E2 -21731.469} C_VEL
LIN {X 0,Y 214.636,Z 776.114,A -85,B 0,C 180,E1 -21733.258,E2 -21733.258} C_VEL
LIN {X 0,Y 209.541,Z 765.435,A -85,B 0,C 180,E1 -21735.506,E2 -21735.506} C_VEL
LIN {X 0,Y 205.67,Z 758.349,A -85,B 0,C 180,E1 -21737.306,E2 -21737.306} C_VEL
LIN {X 0,Y 202.239,Z 752.169,A -85,B 0,C 180,E1 -21739.067,E2 -21739.067} C_VEL
LIN {X 0,Y 198.269,Z 745.209,A -85,B 0,C 180,E1 -21741.442,E2 -21741.442} C_VEL
LIN {X 0,Y 196.422,Z 739.334,A -85,B 0,C 180,E1 -21745.375,E2 -21745.375} C_VEL
LIN {X 0,Y 194.262,Z 733.321,A -85,B 0,C 180,E1 -21750.251,E2 -21750.251} C_VEL
LIN {X 0,Y 193.749,Z 731.499,A -85,B 0,C 180,E1 -21751.865,E2 -21751.865} C_VEL
LIN {X 0,Y 192.653,Z 728.555,A -85,B 0,C 180,E1 -21755.02,E2 -21755.02} C_VEL
LIN {X 0,Y 192.631,Z 728.479,A -85,B 0,C 180,E1 -21758.602,E2 -21758.602} C_VEL
LIN {X 0,Y 192.76,Z 728.462,A -85,B 0,C 180,E1 -21763.042,E2 -21763.042} C_VEL
LIN {X 0,Y 192.794,Z 728.458,A -85,B 0,C 180,E1 -21767.366,E2 -21767.366} C_VEL
LIN {X 0,Y 193.03,Z 728.425,A -85,B 0,C 180,E1 -21771.626,E2 -21771.626} C_VEL
LIN {X 0,Y 193.253,Z 728.413,A -85,B 0,C 180,E1 -21777.916,E2 -21777.916} C_VEL
LIN {X 0,Y 193.433,Z 728.375,A -85,B 0,C 180,E1 -21780,E2 -21780} C_VEL
LIN {X 0,Y 192.966,Z 728.435,A -85,B 0,C 180,E1 -21784.178,E2 -21784.178} C_VEL
LIN {X 0,Y 193.051,Z 728.426,A -85,B 0,C 180,E1 -21788.374,E2 -21788.374} C_VEL
LIN {X 0,Y 192.935,Z 728.714,A -85,B 0,C 180,E1 -21791.358,E2 -21791.358} C_VEL
LIN {X 0,Y 193.168,Z 729.83,A -85,B 0,C 180,E1 -21792.009,E2 -21792.009} C_VEL
LIN {X 0,Y 194.408,Z 732.173,A -85,B 0,C 180,E1 -21792.926,E2 -21792.926} C_VEL
LIN {X 0,Y 197.116,Z 734.381,A -85,B 0,C 180,E1 -21794.519,E2 -21794.519} C_VEL
LIN {X 0,Y 199.139,Z 737.713,A -85,B 0,C 180,E1 -21795.742,E2 -21795.742} C_VEL
LIN {X 0,Y 201.166,Z 739.759,A -85,B 0,C 180,E1 -21796.806,E2 -21796.806} C_VEL
LIN {X 0,Y 203.656,Z 743.33,A -85,B 0,C 180,E1 -21798.095,E2 -21798.095} C_VEL
LIN {X 0,Y 205.066,Z 745.142,A -85,B 0,C 180,E1 -21798.779,E2 -21798.779} C_VEL
LIN {X 0,Y 210.795,Z 753.154,A -85,B 0,C 180,E1 -21801.377,E2 -21801.377} C_VEL
LIN {X 0,Y 217.443,Z 763.627,A -85,B 0,C 180,E1 -21804.083,E2 -21804.083} C_VEL
LIN {X 0,Y 224.015,Z 775.511,A -85,B 0,C 180,E1 -21806.497,E2 -21806.497} C_VEL
LIN {X 0,Y 225.948,Z 779.515,A -85,B 0,C 180,E1 -21807.186,E2 -21807.186} C_VEL
LIN {X 0,Y 224.425,Z 817.565,A -85,B 0,C 180,E1 -21808.65,E2 -21808.65} C_VEL
LIN {X 0,Y 223.369,Z 830.916,A -85,B 0,C 180,E1 -21809.539,E2 -21809.539} C_VEL
LIN {X 0,Y 221.855,Z 842.238,A -85,B 0,C 180,E1 -21810.586,E2 -21810.586} C_VEL
LIN {X 0,Y 219.616,Z 853.988,A -85,B 0,C 180,E1 -21812.007,E2 -21812.007} C_VEL
LIN {X 0,Y 216.809,Z 865.576,A -85,B 0,C 180,E1 -21813.856,E2 -21813.856} C_VEL
LIN {X 0,Y 213.734,Z 875.86,A -85,B 0,C 180,E1 -21815.934,E2 -21815.934} C_VEL
LIN {X 0,Y 210.446,Z 885.075,A -85,B 0,C 180,E1 -21818.303,E2 -21818.303} C_VEL
LIN {X 0,Y 207.086,Z 893.401,A -85,B 0,C 180,E1 -21821.028,E2 -21821.028} C_VEL
LIN {X 0,Y 204.201,Z 899.865,A -85,B 0,C 180,E1 -21823.722,E2 -21823.722} C_VEL
LIN {X 0,Y 201.445,Z 905.486,A -85,B 0,C 180,E1 -21826.714,E2 -21826.714} C_VEL
LIN {X 0,Y 199.374,Z 909.241,A -85,B 0,C 180,E1 -21829.302,E2 -21829.302} C_VEL
LIN {X 0,Y 197.188,Z 912.919,A -85,B 0,C 180,E1 -21832.711,E2 -21832.711} C_VEL
LIN {X 0,Y 195.79,Z 915.018,A -85,B 0,C 180,E1 -21835.65,E2 -21835.65} C_VEL
LIN {X 0,Y 194.42,Z 916.532,A -85,B 0,C 180,E1 -21839.601,E2 -21839.601} C_VEL
LIN {X 0,Y 193.9,Z 916.744,A -85,B 0,C 180,E1 -21841.892,E2 -21841.892} C_VEL
LIN {X 0,Y 193.569,Z 916.223,A -85,B 0,C 180,E1 -21845.189,E2 -21845.189} C_VEL
LIN {X 0,Y 193.655,Z 914.584,A -85,B 0,C 180,E1 -21848.724,E2 -21848.724} C_VEL
LIN {X 0,Y 194.233,Z 911.923,A -85,B 0,C 180,E1 -21852.091,E2 -21852.091} C_VEL
LIN {X 0,Y 195.306,Z 908.146,A -85,B 0,C 180,E1 -21855.414,E2 -21855.414} C_VEL
LIN {X 0,Y 196.664,Z 903.2,A -85,B 0,C 180,E1 -21858.668,E2 -21858.668} C_VEL
LIN {X 0,Y 198.663,Z 896.291,A -85,B 0,C 180,E1 -21862.118,E2 -21862.118} C_VEL
LIN {X 0,Y 200.67,Z 889.02,A -85,B 0,C 180,E1 -21864.98,E2 -21864.98} C_VEL
LIN {X 0,Y 202.756,Z 881.019,A -85,B 0,C 180,E1 -21867.52,E2 -21867.52} C_VEL
LIN {X 0,Y 205.111,Z 871.227,A -85,B 0,C 180,E1 -21870.003,E2 -21870.003} C_VEL
LIN {X 0,Y 207.305,Z 860.428,A -85,B 0,C 180,E1 -21872.189,E2 -21872.189} C_VEL
LIN {X 0,Y 209.206,Z 849.982,A -85,B 0,C 180,E1 -21873.855,E2 -21873.855} C_VEL
LIN {X 0,Y 210.957,Z 837.68,A -85,B 0,C 180,E1 -21875.379,E2 -21875.379} C_VEL
LIN {X 0,Y 212.216,Z 824.318,A -85,B 0,C 180,E1 -21876.6,E2 -21876.6} C_VEL
LIN {X 0,Y 212.924,Z 811.109,A -85,B 0,C 180,E1 -21877.411,E2 -21877.411} C_VEL
LIN {X 0,Y 213.932,Z 776.346,A -85,B 0,C 180,E1 -21878.685,E2 -21878.685} C_VEL
LIN {X 0,Y 214.063,Z 769.591,A -85,B 0,C 180,E1 -21878.936,E2 -21878.936} C_VEL
LIN {X 0,Y 203.539,Z 747.885,A -85,B 0,C 180,E1 -21881.61,E2 -21881.61} C_VEL
LIN {X 0,Y 196.353,Z 735.503,A -85,B 0,C 180,E1 -21883.509,E2 -21883.509} C_VEL
LIN {X 0,Y 193.976,Z 731.595,A -85,B 0,C 180,E1 -21884.167,E2 -21884.167} C_VEL
LIN {X 0,Y 192.844,Z 729.02,A -85,B 0,C 180,E1 -21884.662,E2 -21884.662} C_VEL
LIN {X 0,Y 192.733,Z 728.481,A -85,B 0,C 180,E1 -21885.333,E2 -21885.333} C_VEL
LIN {X 0,Y 192.63,Z 728.469,A -85,B 0,C 180,E1 -21889.172,E2 -21889.172} C_VEL
LIN {X 0,Y 192.625,Z 728.48,A -85,B 0,C 180,E1 -21894.196,E2 -21894.196} C_VEL
LIN {X 0,Y 192.601,Z 728.48,A -85,B 0,C 180,E1 -21898.864,E2 -21898.864} C_VEL
LIN {X 0,Y 192.601,Z 728.459,A -85,B 0,C 180,E1 -21903.189,E2 -21903.189} C_VEL
LIN {X 0,Y 192.549,Z 728.492,A -85,B 0,C 180,E1 -21908.356,E2 -21908.356} C_VEL
LIN {X 0,Y 192.492,Z 728.508,A -85,B 0,C 180,E1 -21913.095,E2 -21913.095} C_VEL
LIN {X 0,Y 192.586,Z 728.671,A -85,B 0,C 180,E1 -21916.477,E2 -21916.477} C_VEL
LIN {X 0,Y 192.812,Z 729.602,A -85,B 0,C 180,E1 -21916.807,E2 -21916.807} C_VEL
LIN {X 0,Y 202.949,Z 759.203,A -85,B 0,C 180,E1 -21919.284,E2 -21919.284} C_VEL
LIN {X 0,Y 200.945,Z 809.576,A -85,B 0,C 180,E1 -21921.983,E2 -21921.983} C_VEL
LIN {X 0,Y 200.438,Z 820.002,A -85,B 0,C 180,E1 -21922.782,E2 -21922.782} C_VEL
LIN {X 0,Y 199.652,Z 830.651,A -85,B 0,C 180,E1 -21923.843,E2 -21923.843} C_VEL
LIN {X 0,Y 198.777,Z 840.584,A -85,B 0,C 180,E1 -21925.079,E2 -21925.079} C_VEL
LIN {X 0,Y 197.797,Z 850.472,A -85,B 0,C 180,E1 -21926.582,E2 -21926.582} C_VEL
LIN {X 0,Y 196.761,Z 860.304,A -85,B 0,C 180,E1 -21928.391,E2 -21928.391} C_VEL
LIN {X 0,Y 195.753,Z 869.5,A -85,B 0,C 180,E1 -21930.418,E2 -21930.418} C_VEL
LIN {X 0,Y 194.752,Z 877.881,A -85,B 0,C 180,E1 -21932.605,E2 -21932.605} C_VEL
LIN {X 0,Y 193.99,Z 885.407,A -85,B 0,C 180,E1 -21934.927,E2 -21934.927} C_VEL
LIN {X 0,Y 193.464,Z 891.239,A -85,B 0,C 180,E1 -21937.013,E2 -21937.013} C_VEL
LIN {X 0,Y 192.972,Z 897.678,A -85,B 0,C 180,E1 -21939.757,E2 -21939.757} C_VEL
LIN {X 0,Y 192.779,Z 902.574,A -85,B 0,C 180,E1 -21942.215,E2 -21942.215} C_VEL
LIN {X 0,Y 192.848,Z 907.477,A -85,B 0,C 180,E1 -21945.22,E2 -21945.22} C_VEL
LIN {X 0,Y 193.422,Z 912.012,A -85,B 0,C 180,E1 -21948.841,E2 -21948.841} C_VEL
LIN {X 0,Y 194.252,Z 914.699,A -85,B 0,C 180,E1 -21951.679,E2 -21951.679} C_VEL
LIN {X 0,Y 195.169,Z 916.225,A -85,B 0,C 180,E1 -21953.798,E2 -21953.798} C_VEL
LIN {X 0,Y 197.035,Z 917.699,A -85,B 0,C 180,E1 -21957.157,E2 -21957.157} C_VEL
LIN {X 0,Y 199.089,Z 918.049,A -85,B 0,C 180,E1 -21960,E2 -21960} C_VEL
LIN {X 0,Y 202.721,Z 917.111,A -85,B 0,C 180,E1 -21963.976,E2 -21963.976} C_VEL
LIN {X 0,Y 204.943,Z 916.001,A -85,B 0,C 180,E1 -21965.997,E2 -21965.997} C_VEL
LIN {X 0,Y 209.66,Z 912.539,A -85,B 0,C 180,E1 -21969.648,E2 -21969.648} C_VEL
LIN {X 0,Y 213.853,Z 908.667,A -85,B 0,C 180,E1 -21972.334,E2 -21972.334} C_VEL
LIN {X 0,Y 218.316,Z 903.654,A -85,B 0,C 180,E1 -21974.924,E2 -21974.924} C_VEL
LIN {X 0,Y 222.392,Z 898.532,A -85,B 0,C 180,E1 -21976.997,E2 -21976.997} C_VEL
LIN {X 0,Y 226.711,Z 892.332,A -85,B 0,C 180,E1 -21978.996,E2 -21978.996} C_VEL
LIN {X 0,Y 231.152,Z 884.99,A -85,B 0,C 180,E1 -21980.931,E2 -21980.931} C_VEL
LIN {X 0,Y 234.906,Z 878.057,A -85,B 0,C 180,E1 -21982.424,E2 -21982.424} C_VEL
LIN {X 0,Y 239.036,Z 869.132,A -85,B 0,C 180,E1 -21984.007,E2 -21984.007} C_VEL
LIN {X 0,Y 242.549,Z 860.511,A -85,B 0,C 180,E1 -21985.256,E2 -21985.256} C_VEL
LIN {X 0,Y 245.569,Z 851.666,A -85,B 0,C 180,E1 -21986.334,E2 -21986.334} C_VEL
LIN {X 0,Y 247.94,Z 843.3,A -85,B 0,C 180,E1 -21987.198,E2 -21987.198} C_VEL
LIN {X 0,Y 250.592,Z 831.633,A -85,B 0,C 180,E1 -21988.15,E2 -21988.15} C_VEL
LIN {X 0,Y 253.595,Z 813.932,A -85,B 0,C 180,E1 -21989.22,E2 -21989.22} C_VEL
LIN {X 0,Y 255.454,Z 802.707,A -85,B 0,C 180,E1 -21989.81,E2 -21989.81} C_VEL
LIN {X 0,Y 254.442,Z 800.142,A -85,B 0,C 180,E1 -21991.367,E2 -21991.367} C_VEL
LIN {X 0,Y 253.826,Z 798.425,A -85,B 0,C 180,E1 -21992.612,E2 -21992.612} C_VEL
LIN {X 0,Y 253.035,Z 796.486,A -85,B 0,C 180,E1 -21995.035,E2 -21995.035} C_VEL
LIN {X 0,Y 252.678,Z 796.61,A -85,B 0,C 180,E1 -21997.236,E2 -21997.236} C_VEL
LIN {X 0,Y 252.623,Z 797.023,A -85,B 0,C 180,E1 -21998.058,E2 -21998.058} C_VEL
LIN {X 0,Y 252.58,Z 798.134,A -85,B 0,C 180,E1 -21998.91,E2 -21998.91} C_VEL
LIN {X 0,Y 252.371,Z 800.229,A -85,B 0,C 180,E1 -21999.675,E2 -21999.675} C_VEL
LIN {X 0,Y 251.742,Z 805.951,A -85,B 0,C 180,E1 -22001.015,E2 -22001.015} C_VEL
LIN {X 0,Y 251.401,Z 809.945,A -85,B 0,C 180,E1 -22001.899,E2 -22001.899} C_VEL
LIN {X 0,Y 249.943,Z 820.406,A -85,B 0,C 180,E1 -22003.02,E2 -22003.02} C_VEL
LIN {X 0,Y 247.649,Z 836.669,A -85,B 0,C 180,E1 -22004.481,E2 -22004.481} C_VEL
LIN {X 0,Y 245.061,Z 852.125,A -85,B 0,C 180,E1 -22005.586,E2 -22005.586} C_VEL
LIN {X 0,Y 240.553,Z 868.05,A -85,B 0,C 180,E1 -22006.493,E2 -22006.493} C_VEL
LIN {X 0,Y 236.128,Z 880.183,A -85,B 0,C 180,E1 -22007.378,E2 -22007.378} C_VEL
LIN {X 0,Y 231.481,Z 890.978,A -85,B 0,C 180,E1 -22008.38,E2 -22008.38} C_VEL
LIN {X 0,Y 227.06,Z 900.057,A -85,B 0,C 180,E1 -22009.456,E2 -22009.456} C_VEL
LIN {X 0,Y 221.618,Z 910.089,A -85,B 0,C 180,E1 -22010.926,E2 -22010.926} C_VEL
LIN {X 0,Y 216.566,Z 918.627,A -85,B 0,C 180,E1 -22012.518,E2 -22012.518} C_VEL
LIN {X 0,Y 211.247,Z 926.799,A -85,B 0,C 180,E1 -22014.391,E2 -22014.391} C_VEL
LIN {X 0,Y 206.347,Z 933.868,A -85,B 0,C 180,E1 -22016.392,E2 -22016.392} C_VEL
LIN {X 0,Y 201.938,Z 939.959,A -85,B 0,C 180,E1 -22018.528,E2 -22018.528} C_VEL
LIN {X 0,Y 197.226,Z 946.185,A -85,B 0,C 180,E1 -22021.242,E2 -22021.242} C_VEL
LIN {X 0,Y 193.211,Z 951.343,A -85,B 0,C 180,E1 -22024.116,E2 -22024.116} C_VEL
LIN {X 0,Y 189.97,Z 955.58,A -85,B 0,C 180,E1 -22027.139,E2 -22027.139} C_VEL
LIN {X 0,Y 187.422,Z 958.929,A -85,B 0,C 180,E1 -22030.273,E2 -22030.273} C_VEL
LIN {X 0,Y 185.299,Z 962.054,A -85,B 0,C 180,E1 -22034.6,E2 -22034.6} C_VEL
LIN {X 0,Y 184.553,Z 963.768,A -85,B 0,C 180,E1 -22039.02,E2 -22039.02} C_VEL
LIN {X 0,Y 184.586,Z 964.319,A -85,B 0,C 180,E1 -22040.684,E2 -22040.684} C_VEL
LIN {X 0,Y 184.717,Z 966.945,A -85,B 0,C 180,E1 -22043.443,E2 -22043.443} C_VEL
LIN {X 0,Y 185.033,Z 968.56,A -85,B 0,C 180,E1 -22045.64,E2 -22045.64} C_VEL
LIN {X 0,Y 185.289,Z 969.687,A -85,B 0,C 180,E1 -22047.823,E2 -22047.823} C_VEL
LIN {X 0,Y 185.604,Z 970.346,A -85,B 0,C 180,E1 -22049.997,E2 -22049.997} C_VEL
LIN {X 0,Y 185.23,Z 970.476,A -85,B 0,C 180,E1 -22052.171,E2 -22052.171} C_VEL
LIN {X 0,Y 184.87,Z 970.186,A -85,B 0,C 180,E1 -22054.357,E2 -22054.357} C_VEL
LIN {X 0,Y 184.374,Z 968.927,A -85,B 0,C 180,E1 -22057.662,E2 -22057.662} C_VEL
LIN {X 0,Y 184.325,Z 966.759,A -85,B 0,C 180,E1 -22060.987,E2 -22060.987} C_VEL
LIN {X 0,Y 184.902,Z 963.669,A -85,B 0,C 180,E1 -22064.3,E2 -22064.3} C_VEL
LIN {X 0,Y 186.107,Z 959.589,A -85,B 0,C 180,E1 -22067.581,E2 -22067.581} C_VEL
LIN {X 0,Y 188.17,Z 954.113,A -85,B 0,C 180,E1 -22070.976,E2 -22070.976} C_VEL
LIN {X 0,Y 191.268,Z 946.931,A -85,B 0,C 180,E1 -22074.413,E2 -22074.413} C_VEL
LIN {X 0,Y 194.726,Z 938.877,A -85,B 0,C 180,E1 -22077.394,E2 -22077.394} C_VEL
LIN {X 0,Y 198.856,Z 928.928,A -85,B 0,C 180,E1 -22080.236,E2 -22080.236} C_VEL
LIN {X 0,Y 202.836,Z 918.757,A -85,B 0,C 180,E1 -22082.48,E2 -22082.48} C_VEL
LIN {X 0,Y 206.75,Z 907.354,A -85,B 0,C 180,E1 -22084.407,E2 -22084.407} C_VEL
LIN {X 0,Y 209.975,Z 896.284,A -85,B 0,C 180,E1 -22085.851,E2 -22085.851} C_VEL
LIN {X 0,Y 212.883,Z 883.666,A -85,B 0,C 180,E1 -22087.11,E2 -22087.11} C_VEL
LIN {X 0,Y 215.166,Z 870.48,A -85,B 0,C 180,E1 -22088.022,E2 -22088.022} C_VEL
LIN {X 0,Y 216.639,Z 856.513,A -85,B 0,C 180,E1 -22088.652,E2 -22088.652} C_VEL
LIN {X 0,Y 217.377,Z 842.261,A -85,B 0,C 180,E1 -22089.155,E2 -22089.155} C_VEL
LIN {X 0,Y 216.512,Z 819.845,A -85,B 0,C 180,E1 -22090.478,E2 -22090.478} C_VEL
LIN {X 0,Y 215.302,Z 800.164,A -85,B 0,C 180,E1 -22091.806,E2 -22091.806} C_VEL
LIN {X 0,Y 214.193,Z 789.536,A -85,B 0,C 180,E1 -22092.677,E2 -22092.677} C_VEL
LIN {X 0,Y 210.054,Z 779.356,A -85,B 0,C 180,E1 -22094.535,E2 -22094.535} C_VEL
LIN {X 0,Y 205.499,Z 769.667,A -85,B 0,C 180,E1 -22096.675,E2 -22096.675} C_VEL
LIN {X 0,Y 202.146,Z 763.253,A -85,B 0,C 180,E1 -22098.371,E2 -22098.371} C_VEL
LIN {X 0,Y 198.841,Z 757.143,A -85,B 0,C 180,E1 -22100.188,E2 -22100.188} C_VEL
LIN {X 0,Y 194.86,Z 750.376,A -85,B 0,C 180,E1 -22102.566,E2 -22102.566} C_VEL
LIN {X 0,Y 190.315,Z 742.727,A -85,B 0,C 180,E1 -22105.84,E2 -22105.84} C_VEL
LIN {X 0,Y 188.521,Z 737.598,A -85,B 0,C 180,E1 -22110.014,E2 -22110.014} C_VEL
LIN {X 0,Y 187.818,Z 735.338,A -85,B 0,C 180,E1 -22112.113,E2 -22112.113} C_VEL
LIN {X 0,Y 186.58,Z 732.189,A -85,B 0,C 180,E1 -22115.522,E2 -22115.522} C_VEL
LIN {X 0,Y 185.588,Z 729.433,A -85,B 0,C 180,E1 -22119.206,E2 -22119.206} C_VEL
LIN {X 0,Y 185.706,Z 729.341,A -85,B 0,C 180,E1 -22122.377,E2 -22122.377} C_VEL
LIN {X 0,Y 185.72,Z 729.338,A -85,B 0,C 180,E1 -22126.877,E2 -22126.877} C_VEL
LIN {X 0,Y 185.976,Z 729.303,A -85,B 0,C 180,E1 -22131.306,E2 -22131.306} C_VEL
LIN {X 0,Y 186.196,Z 729.29,A -85,B 0,C 180,E1 -22137.837,E2 -22137.837} C_VEL
LIN {X 0,Y 186.396,Z 729.251,A -85,B 0,C 180,E1 -22140,E2 -22140} C_VEL
LIN {X 0,Y 185.941,Z 729.362,A -85,B 0,C 180,E1 -22145.967,E2 -22145.967} C_VEL
LIN {X 0,Y 186.035,Z 729.906,A -85,B 0,C 180,E1 -22147.053,E2 -22147.053} C_VEL
LIN {X 0,Y 187.697,Z 733.146,A -85,B 0,C 180,E1 -22148.887,E2 -22148.887} C_VEL
LIN {X 0,Y 190.516,Z 735.475,A -85,B 0,C 180,E1 -22150.965,E2 -22150.965} C_VEL
LIN {X 0,Y 192.256,Z 738.564,A -85,B 0,C 180,E1 -22152.268,E2 -22152.268} C_VEL
LIN {X 0,Y 194.775,Z 740.921,A -85,B 0,C 180,E1 -22153.833,E2 -22153.833} C_VEL
LIN {X 0,Y 197.011,Z 744.257,A -85,B 0,C 180,E1 -22155.207,E2 -22155.207} C_VEL
LIN {X 0,Y 198.461,Z 745.827,A -85,B 0,C 180,E1 -22156.012,E2 -22156.012} C_VEL
LIN {X 0,Y 201.273,Z 749.728,A -85,B 0,C 180,E1 -22157.533,E2 -22157.533} C_VEL
LIN {X 0,Y 207.627,Z 758.906,A -85,B 0,C 180,E1 -22160.612,E2 -22160.612} C_VEL
LIN {X 0,Y 213.777,Z 768.829,A -85,B 0,C 180,E1 -22163.236,E2 -22163.236} C_VEL
LIN {X 0,Y 220.015,Z 780.426,A -85,B 0,C 180,E1 -22165.668,E2 -22165.668} C_VEL
LIN {X 0,Y 220.901,Z 782.332,A -85,B 0,C 180,E1 -22166.003,E2 -22166.003} C_VEL
LIN {X 0,Y 219.361,Z 816.976,A -85,B 0,C 180,E1 -22167.333,E2 -22167.333} C_VEL
LIN {X 0,Y 218.378,Z 829.721,A -85,B 0,C 180,E1 -22168.143,E2 -22168.143} C_VEL
LIN {X 0,Y 216.765,Z 841.82,A -85,B 0,C 180,E1 -22169.24,E2 -22169.24} C_VEL
LIN {X 0,Y 214.469,Z 853.764,A -85,B 0,C 180,E1 -22170.668,E2 -22170.668} C_VEL
LIN {X 0,Y 211.876,Z 864.17,A -85,B 0,C 180,E1 -22172.27,E2 -22172.27} C_VEL
LIN {X 0,Y 208.664,Z 874.835,A -85,B 0,C 180,E1 -22174.376,E2 -22174.376} C_VEL
LIN {X 0,Y 205.523,Z 883.572,A -85,B 0,C 180,E1 -22176.53,E2 -22176.53} C_VEL
LIN {X 0,Y 202.049,Z 892.171,A -85,B 0,C 180,E1 -22179.21,E2 -22179.21} C_VEL
LIN {X 0,Y 198.428,Z 899.836,A -85,B 0,C 180,E1 -22182.296,E2 -22182.296} C_VEL
LIN {X 0,Y 195.48,Z 905.692,A -85,B 0,C 180,E1 -22185.395,E2 -22185.395} C_VEL
LIN {X 0,Y 192.545,Z 910.751,A -85,B 0,C 180,E1 -22188.932,E2 -22188.932} C_VEL
LIN {X 0,Y 190.92,Z 913.211,A -85,B 0,C 180,E1 -22191.264,E2 -22191.264} C_VEL
LIN {X 0,Y 189.066,Z 915.899,A -85,B 0,C 180,E1 -22194.865,E2 -22194.865} C_VEL
LIN {X 0,Y 187.378,Z 917.623,A -85,B 0,C 180,E1 -22199.618,E2 -22199.618} C_VEL
LIN {X 0,Y 186.68,Z 917.655,A -85,B 0,C 180,E1 -22203.147,E2 -22203.147} C_VEL
LIN {X 0,Y 186.548,Z 917.098,A -85,B 0,C 180,E1 -22205.521,E2 -22205.521} C_VEL
LIN {X 0,Y 186.572,Z 916.063,A -85,B 0,C 180,E1 -22207.875,E2 -22207.875} C_VEL
LIN {X 0,Y 186.82,Z 914.561,A -85,B 0,C 180,E1 -22210.214,E2 -22210.214} C_VEL
LIN {X 0,Y 187.629,Z 911.413,A -85,B 0,C 180,E1 -22213.688,E2 -22213.688} C_VEL
LIN {X 0,Y 188.899,Z 907.125,A -85,B 0,C 180,E1 -22217.104,E2 -22217.104} C_VEL
LIN {X 0,Y 190.474,Z 901.626,A -85,B 0,C 180,E1 -22220.446,E2 -22220.446} C_VEL
LIN {X 0,Y 192.552,Z 894.643,A -85,B 0,C 180,E1 -22223.717,E2 -22223.717} C_VEL
LIN {X 0,Y 195.008,Z 885.991,A -85,B 0,C 180,E1 -22226.904,E2 -22226.904} C_VEL
LIN {X 0,Y 197.467,Z 876.533,A -85,B 0,C 180,E1 -22229.64,E2 -22229.64} C_VEL
LIN {X 0,Y 199.837,Z 866.184,A -85,B 0,C 180,E1 -22232.018,E2 -22232.018} C_VEL
LIN {X 0,Y 202.047,Z 855.319,A -85,B 0,C 180,E1 -22233.992,E2 -22233.992} C_VEL
LIN {X 0,Y 204.027,Z 843.236,A -85,B 0,C 180,E1 -22235.686,E2 -22235.686} C_VEL
LIN {X 0,Y 205.481,Z 830.887,A -85,B 0,C 180,E1 -22237.002,E2 -22237.002} C_VEL
LIN {X 0,Y 206.422,Z 817.778,A -85,B 0,C 180,E1 -22238.004,E2 -22238.004} C_VEL
LIN {X 0,Y 206.89,Z 801.623,A -85,B 0,C 180,E1 -22238.747,E2 -22238.747} C_VEL
LIN {X 0,Y 207.896,Z 771.629,A -85,B 0,C 180,E1 -22239.838,E2 -22239.838} C_VEL
LIN {X 0,Y 198.217,Z 751.658,A -85,B 0,C 180,E1 -22242.419,E2 -22242.419} C_VEL
LIN {X 0,Y 191.326,Z 739.705,A -85,B 0,C 180,E1 -22244.332,E2 -22244.332} C_VEL
LIN {X 0,Y 187.204,Z 732.925,A -85,B 0,C 180,E1 -22245.548,E2 -22245.548} C_VEL
LIN {X 0,Y 185.762,Z 729.975,A -85,B 0,C 180,E1 -22246.153,E2 -22246.153} C_VEL
LIN {X 0,Y 185.683,Z 729.383,A -85,B 0,C 180,E1 -22246.778,E2 -22246.778} C_VEL
LIN {X 0,Y 185.552,Z 729.365,A -85,B 0,C 180,E1 -22252.26,E2 -22252.26} C_VEL
LIN {X 0,Y 185.498,Z 729.346,A -85,B 0,C 180,E1 -22257.046,E2 -22257.046} C_VEL
LIN {X 0,Y 185.536,Z 729.357,A -85,B 0,C 180,E1 -22262.03,E2 -22262.03} C_VEL
LIN {X 0,Y 185.507,Z 729.351,A -85,B 0,C 180,E1 -22267.317,E2 -22267.317} C_VEL
LIN {X 0,Y 185.469,Z 729.382,A -85,B 0,C 180,E1 -22270.723,E2 -22270.723} C_VEL
LIN {X 0,Y 185.56,Z 729.599,A -85,B 0,C 180,E1 -22275.954,E2 -22275.954} C_VEL
LIN {X 0,Y 185.802,Z 730.625,A -85,B 0,C 180,E1 -22276.278,E2 -22276.278} C_VEL
LIN {X 0,Y 195.938,Z 760.455,A -85,B 0,C 180,E1 -22278.876,E2 -22278.876} C_VEL
LIN {X 0,Y 193.924,Z 811.084,A -85,B 0,C 180,E1 -22281.72,E2 -22281.72} C_VEL
LIN {X 0,Y 193.307,Z 821.833,A -85,B 0,C 180,E1 -22282.587,E2 -22282.587} C_VEL
LIN {X 0,Y 192.454,Z 832.771,A -85,B 0,C 180,E1 -22283.741,E2 -22283.741} C_VEL
LIN {X 0,Y 191.615,Z 842.569,A -85,B 0,C 180,E1 -22285.033,E2 -22285.033} C_VEL
LIN {X 0,Y 190.679,Z 851.452,A -85,B 0,C 180,E1 -22286.436,E2 -22286.436} C_VEL
LIN {X 0,Y 189.685,Z 861.02,A -85,B 0,C 180,E1 -22288.249,E2 -22288.249} C_VEL
LIN {X 0,Y 188.731,Z 869.392,A -85,B 0,C 180,E1 -22290.128,E2 -22290.128} C_VEL
LIN {X 0,Y 187.823,Z 876.958,A -85,B 0,C 180,E1 -22292.113,E2 -22292.113} C_VEL
LIN {X 0,Y 187.028,Z 884.443,A -85,B 0,C 180,E1 -22294.409,E2 -22294.409} C_VEL
LIN {X 0,Y 186.313,Z 892.195,A -85,B 0,C 180,E1 -22297.254,E2 -22297.254} C_VEL
LIN {X 0,Y 185.867,Z 898.688,A -85,B 0,C 180,E1 -22300.104,E2 -22300.104} C_VEL
LIN {X 0,Y 185.677,Z 903.161,A -85,B 0,C 180,E1 -22302.373,E2 -22302.373} C_VEL
LIN {X 0,Y 185.818,Z 908.582,A -85,B 0,C 180,E1 -22305.768,E2 -22305.768} C_VEL
LIN {X 0,Y 186.422,Z 912.758,A -85,B 0,C 180,E1 -22309.135,E2 -22309.135} C_VEL
LIN {X 0,Y 187.052,Z 914.971,A -85,B 0,C 180,E1 -22311.356,E2 -22311.356} C_VEL
LIN {X 0,Y 189.076,Z 918.003,A -85,B 0,C 180,E1 -22315.736,E2 -22315.736} C_VEL
LIN {X 0,Y 190.388,Z 918.876,A -85,B 0,C 180,E1 -22317.884,E2 -22317.884} C_VEL
LIN {X 0,Y 191.939,Z 919.328,A -85,B 0,C 180,E1 -22320,E2 -22320} C_VEL
LIN {X 0,Y 195.69,Z 918.891,A -85,B 0,C 180,E1 -22324.119,E2 -22324.119} C_VEL
LIN {X 0,Y 200.26,Z 916.846,A -85,B 0,C 180,E1 -22328.069,E2 -22328.069} C_VEL
LIN {X 0,Y 204.229,Z 914.159,A -85,B 0,C 180,E1 -22330.91,E2 -22330.91} C_VEL
LIN {X 0,Y 208.721,Z 910.36,A -85,B 0,C 180,E1 -22333.633,E2 -22333.633} C_VEL
LIN {X 0,Y 213.488,Z 905.5,A -85,B 0,C 180,E1 -22336.249,E2 -22336.249} C_VEL
LIN {X 0,Y 218.676,Z 899.311,A -85,B 0,C 180,E1 -22338.747,E2 -22338.747} C_VEL
LIN {X 0,Y 223.315,Z 893.056,A -85,B 0,C 180,E1 -22340.735,E2 -22340.735} C_VEL
LIN {X 0,Y 227.117,Z 887.222,A -85,B 0,C 180,E1 -22342.276,E2 -22342.276} C_VEL
LIN {X 0,Y 231.515,Z 879.641,A -85,B 0,C 180,E1 -22343.923,E2 -22343.923} C_VEL
LIN {X 0,Y 235.897,Z 870.869,A -85,B 0,C 180,E1 -22345.489,E2 -22345.489} C_VEL
LIN {X 0,Y 239.747,Z 861.853,A -85,B 0,C 180,E1 -22346.789,E2 -22346.789} C_VEL
LIN {X 0,Y 242.85,Z 853.423,A -85,B 0,C 180,E1 -22347.817,E2 -22347.817} C_VEL
LIN {X 0,Y 245.392,Z 845.203,A -85,B 0,C 180,E1 -22348.667,E2 -22348.667} C_VEL
LIN {X 0,Y 248.222,Z 833.478,A -85,B 0,C 180,E1 -22349.625,E2 -22349.625} C_VEL
LIN {X 0,Y 251.54,Z 815.499,A -85,B 0,C 180,E1 -22350.718,E2 -22350.718} C_VEL
LIN {X 0,Y 252.92,Z 807.623,A -85,B 0,C 180,E1 -22351.156,E2 -22351.156} C_VEL
LIN {X 0,Y 252.112,Z 805.203,A -85,B 0,C 180,E1 -22352.861,E2 -22352.861} C_VEL
LIN {X 0,Y 251.394,Z 803.348,A -85,B 0,C 180,E1 -22355.298,E2 -22355.298} C_VEL
LIN {X 0,Y 251.106,Z 803.527,A -85,B 0,C 180,E1 -22357.15,E2 -22357.15} C_VEL
LIN {X 0,Y 251.303,Z 805.217,A -85,B 0,C 180,E1 -22359.895,E2 -22359.895} C_VEL
LIN {X 0,Y 251.568,Z 807.048,A -85,B 0,C 180,E1 -22361.153,E2 -22361.153} C_VEL
LIN {X 0,Y 251.401,Z 809.945,A -85,B 0,C 180,E1 -22361.899,E2 -22361.899} C_VEL
LIN {X 0,Y 251.106,Z 812.978,A -85,B 0,C 180,E1 -22362.422,E2 -22362.422} C_VEL
LIN {X 0,Y 250.41,Z 817.468,A -85,B 0,C 180,E1 -22362.797,E2 -22362.797} C_VEL
LIN {X 0,Y 249.003,Z 824.213,A -85,B 0,C 180,E1 -22362.953,E2 -22362.953} C_VEL
LIN {X 0,Y 246.162,Z 836.563,A -85,B 0,C 180,E1 -22362.946,E2 -22362.946} C_VEL
LIN {X 0,Y 245.368,Z 840.614,A -85,B 0,C 180,E1 -22363.113,E2 -22363.113} C_VEL
LIN {X 0,Y 242.949,Z 852.693,A -85,B 0,C 180,E1 -22364.001,E2 -22364.001} C_VEL
LIN {X 0,Y 238.728,Z 866.465,A -85,B 0,C 180,E1 -22364.784,E2 -22364.784} C_VEL
LIN {X 0,Y 234.566,Z 877.485,A -85,B 0,C 180,E1 -22365.541,E2 -22365.541} C_VEL
LIN {X 0,Y 229.739,Z 888.322,A -85,B 0,C 180,E1 -22366.501,E2 -22366.501} C_VEL
LIN {X 0,Y 224.419,Z 898.714,A -85,B 0,C 180,E1 -22367.674,E2 -22367.674} C_VEL
LIN {X 0,Y 219.321,Z 907.651,A -85,B 0,C 180,E1 -22368.932,E2 -22368.932} C_VEL
LIN {X 0,Y 214.556,Z 915.361,A -85,B 0,C 180,E1 -22370.299,E2 -22370.299} C_VEL
LIN {X 0,Y 208.839,Z 923.75,A -85,B 0,C 180,E1 -22372.106,E2 -22372.106} C_VEL
LIN {X 0,Y 203.491,Z 930.995,A -85,B 0,C 180,E1 -22374.043,E2 -22374.043} C_VEL
LIN {X 0,Y 197.744,Z 938.344,A -85,B 0,C 180,E1 -22376.569,E2 -22376.569} C_VEL
LIN {X 0,Y 192.59,Z 944.547,A -85,B 0,C 180,E1 -22379.274,E2 -22379.274} C_VEL
LIN {X 0,Y 188.163,Z 949.709,A -85,B 0,C 180,E1 -22382.164,E2 -22382.164} C_VEL
LIN {X 0,Y 184.461,Z 953.954,A -85,B 0,C 180,E1 -22385.219,E2 -22385.219} C_VEL
LIN {X 0,Y 181.583,Z 957.189,A -85,B 0,C 180,E1 -22388.263,E2 -22388.263} C_VEL
LIN {X 0,Y 179.434,Z 959.845,A -85,B 0,C 180,E1 -22391.736,E2 -22391.736} C_VEL
LIN {X 0,Y 177.841,Z 961.996,A -85,B 0,C 180,E1 -22396.281,E2 -22396.281} C_VEL
LIN {X 0,Y 177.605,Z 962.794,A -85,B 0,C 180,E1 -22400.027,E2 -22400.027} C_VEL
LIN {X 0,Y 177.646,Z 965.767,A -85,B 0,C 180,E1 -22403.18,E2 -22403.18} C_VEL
LIN {X 0,Y 177.953,Z 967.413,A -85,B 0,C 180,E1 -22405.466,E2 -22405.466} C_VEL
LIN {X 0,Y 178.232,Z 968.594,A -85,B 0,C 180,E1 -22407.737,E2 -22407.737} C_VEL
LIN {X 0,Y 178.562,Z 969.29,A -85,B 0,C 180,E1 -22409.997,E2 -22409.997} C_VEL
LIN {X 0,Y 178.166,Z 969.442,A -85,B 0,C 180,E1 -22412.257,E2 -22412.257} C_VEL
LIN {X 0,Y 177.771,Z 969.17,A -85,B 0,C 180,E1 -22414.532,E2 -22414.532} C_VEL
LIN {X 0,Y 177.315,Z 968.07,A -85,B 0,C 180,E1 -22417.74,E2 -22417.74} C_VEL
LIN {X 0,Y 177.304,Z 965.845,A -85,B 0,C 180,E1 -22421.428,E2 -22421.428} C_VEL
LIN {X 0,Y 178.339,Z 961.616,A -85,B 0,C 180,E1 -22426.009,E2 -22426.009} C_VEL
LIN {X 0,Y 179.854,Z 957.256,A -85,B 0,C 180,E1 -22429.395,E2 -22429.395} C_VEL
LIN {X 0,Y 182.811,Z 950.787,A -85,B 0,C 180,E1 -22433.203,E2 -22433.203} C_VEL
LIN {X 0,Y 185.867,Z 943.828,A -85,B 0,C 180,E1 -22436.374,E2 -22436.374} C_VEL
LIN {X 0,Y 189.823,Z 935.335,A -85,B 0,C 180,E1 -22439.374,E2 -22439.374} C_VEL
LIN {X 0,Y 193.494,Z 926.743,A -85,B 0,C 180,E1 -22441.776,E2 -22441.776} C_VEL
LIN {X 0,Y 197.752,Z 916.289,A -85,B 0,C 180,E1 -22444.034,E2 -22444.034} C_VEL
LIN {X 0,Y 201.882,Z 904.604,A -85,B 0,C 180,E1 -22445.973,E2 -22445.973} C_VEL
LIN {X 0,Y 205.272,Z 893.177,A -85,B 0,C 180,E1 -22447.42,E2 -22447.42} C_VEL
LIN {X 0,Y 207.878,Z 882.018,A -85,B 0,C 180,E1 -22448.502,E2 -22448.502} C_VEL
LIN {X 0,Y 210.21,Z 868.513,A -85,B 0,C 180,E1 -22449.433,E2 -22449.433} C_VEL
LIN {X 0,Y 211.669,Z 855.032,A -85,B 0,C 180,E1 -22450.028,E2 -22450.028} C_VEL
LIN {X 0,Y 212.297,Z 842.868,A -85,B 0,C 180,E1 -22450.472,E2 -22450.472} C_VEL
LIN {X 0,Y 211.435,Z 817.076,A -85,B 0,C 180,E1 -22452.044,E2 -22452.044} C_VEL
LIN {X 0,Y 210.224,Z 798.399,A -85,B 0,C 180,E1 -22453.42,E2 -22453.42} C_VEL
LIN {X 0,Y 209.615,Z 792.642,A -85,B 0,C 180,E1 -22453.933,E2 -22453.933} C_VEL
LIN {X 0,Y 205.944,Z 783.381,A -85,B 0,C 180,E1 -22455.696,E2 -22455.696} C_VEL
LIN {X 0,Y 201.695,Z 774.111,A -85,B 0,C 180,E1 -22457.853,E2 -22457.853} C_VEL
LIN {X 0,Y 198.636,Z 768.054,A -85,B 0,C 180,E1 -22459.51,E2 -22459.51} C_VEL
LIN {X 0,Y 195.849,Z 762.679,A -85,B 0,C 180,E1 -22461.15,E2 -22461.15} C_VEL
LIN {X 0,Y 192.091,Z 756.053,A -85,B 0,C 180,E1 -22463.539,E2 -22463.539} C_VEL
LIN {X 0,Y 187.369,Z 748.149,A -85,B 0,C 180,E1 -22467.052,E2 -22467.052} C_VEL
LIN {X 0,Y 181.946,Z 739.26,A -85,B 0,C 180,E1 -22472.386,E2 -22472.386} C_VEL
LIN {X 0,Y 180.275,Z 735.179,A -85,B 0,C 180,E1 -22477.055,E2 -22477.055} C_VEL
LIN {X 0,Y 179.556,Z 733.061,A -85,B 0,C 180,E1 -22479.938,E2 -22479.938} C_VEL
LIN {X 0,Y 178.69,Z 730.296,A -85,B 0,C 180,E1 -22484.897,E2 -22484.897} C_VEL
LIN {X 0,Y 178.903,Z 730.184,A -85,B 0,C 180,E1 -22490.96,E2 -22490.96} C_VEL
LIN {X 0,Y 178.858,Z 730.19,A -85,B 0,C 180,E1 -22495.493,E2 -22495.493} C_VEL
LIN {X 0,Y 179.393,Z 730.349,A -85,B 0,C 180,E1 -22500,E2 -22500} C_VEL
LIN {X 0,Y 179.484,Z 731.426,A -85,B 0,C 180,E1 -22501.262,E2 -22501.262} C_VEL
LIN {X 0,Y 181.022,Z 734.375,A -85,B 0,C 180,E1 -22503.478,E2 -22503.478} C_VEL
LIN {X 0,Y 184.038,Z 736.553,A -85,B 0,C 180,E1 -22506.503,E2 -22506.503} C_VEL
LIN {X 0,Y 186.201,Z 740.082,A -85,B 0,C 180,E1 -22508.547,E2 -22508.547} C_VEL
LIN {X 0,Y 188.376,Z 741.981,A -85,B 0,C 180,E1 -22510.214,E2 -22510.214} C_VEL
LIN {X 0,Y 190.422,Z 745.265,A -85,B 0,C 180,E1 -22511.78,E2 -22511.78} C_VEL
LIN {X 0,Y 192.494,Z 747.426,A -85,B 0,C 180,E1 -22513.147,E2 -22513.147} C_VEL
LIN {X 0,Y 195.154,Z 751.042,A -85,B 0,C 180,E1 -22514.811,E2 -22514.811} C_VEL
LIN {X 0,Y 196.777,Z 753.414,A -85,B 0,C 180,E1 -22515.779,E2 -22515.779} C_VEL
LIN {X 0,Y 199.689,Z 757.521,A -85,B 0,C 180,E1 -22517.39,E2 -22517.39} C_VEL
LIN {X 0,Y 204.404,Z 764.466,A -85,B 0,C 180,E1 -22519.751,E2 -22519.751} C_VEL
LIN {X 0,Y 210.306,Z 774.25,A -85,B 0,C 180,E1 -22522.42,E2 -22522.42} C_VEL
LIN {X 0,Y 215.836,Z 784.914,A -85,B 0,C 180,E1 -22524.722,E2 -22524.722} C_VEL
LIN {X 0,Y 214.262,Z 819.506,A -85,B 0,C 180,E1 -22526.12,E2 -22526.12} C_VEL
LIN {X 0,Y 213.03,Z 832.943,A -85,B 0,C 180,E1 -22527.04,E2 -22527.04} C_VEL
LIN {X 0,Y 211.253,Z 844.862,A -85,B 0,C 180,E1 -22528.19,E2 -22528.19} C_VEL
LIN {X 0,Y 208.749,Z 856.534,A -85,B 0,C 180,E1 -22529.668,E2 -22529.668} C_VEL
LIN {X 0,Y 205.885,Z 867.186,A -85,B 0,C 180,E1 -22531.424,E2 -22531.424} C_VEL
LIN {X 0,Y 202.462,Z 877.582,A -85,B 0,C 180,E1 -22533.587,E2 -22533.587} C_VEL
LIN {X 0,Y 199.21,Z 885.941,A -85,B 0,C 180,E1 -22535.77,E2 -22535.77} C_VEL
LIN {X 0,Y 195.501,Z 894.365,A -85,B 0,C 180,E1 -22538.572,E2 -22538.572} C_VEL
LIN {X 0,Y 191.704,Z 901.974,A -85,B 0,C 180,E1 -22541.837,E2 -22541.837} C_VEL
LIN {X 0,Y 188.578,Z 907.69,A -85,B 0,C 180,E1 -22545.081,E2 -22545.081} C_VEL
LIN {X 0,Y 185.714,Z 912.201,A -85,B 0,C 180,E1 -22548.506,E2 -22548.506} C_VEL
LIN {X 0,Y 183.328,Z 915.582,A -85,B 0,C 180,E1 -22552.171,E2 -22552.171} C_VEL
LIN {X 0,Y 182.106,Z 917.145,A -85,B 0,C 180,E1 -22554.632,E2 -22554.632} C_VEL
LIN {X 0,Y 180.531,Z 918.613,A -85,B 0,C 180,E1 -22558.921,E2 -22558.921} C_VEL
LIN {X 0,Y 179.816,Z 918.792,A -85,B 0,C 180,E1 -22562.034,E2 -22562.034} C_VEL
LIN {X 0,Y 179.547,Z 918.357,A -85,B 0,C 180,E1 -22564.5,E2 -22564.5} C_VEL
LIN {X 0,Y 179.517,Z 917.487,A -85,B 0,C 180,E1 -22566.956,E2 -22566.956} C_VEL
LIN {X 0,Y 179.712,Z 915.866,A -85,B 0,C 180,E1 -22569.814,E2 -22569.814} C_VEL
LIN {X 0,Y 180.731,Z 912.047,A -85,B 0,C 180,E1 -22574.208,E2 -22574.208} C_VEL
LIN {X 0,Y 182.077,Z 907.625,A -85,B 0,C 180,E1 -22577.747,E2 -22577.747} C_VEL
LIN {X 0,Y 183.775,Z 901.948,A -85,B 0,C 180,E1 -22581.204,E2 -22581.204} C_VEL
LIN {X 0,Y 185.972,Z 894.82,A -85,B 0,C 180,E1 -22584.582,E2 -22584.582} C_VEL
LIN {X 0,Y 188.138,Z 887.556,A -85,B 0,C 180,E1 -22587.327,E2 -22587.327} C_VEL
LIN {X 0,Y 190.528,Z 878.83,A -85,B 0,C 180,E1 -22590.003,E2 -22590.003} C_VEL
LIN {X 0,Y 192.895,Z 869.25,A -85,B 0,C 180,E1 -22592.352,E2 -22592.352} C_VEL
LIN {X 0,Y 195.131,Z 858.84,A -85,B 0,C 180,E1 -22594.393,E2 -22594.393} C_VEL
LIN {X 0,Y 197.219,Z 847.493,A -85,B 0,C 180,E1 -22596.14,E2 -22596.14} C_VEL
LIN {X 0,Y 198.801,Z 836.184,A -85,B 0,C 180,E1 -22597.494,E2 -22597.494} C_VEL
LIN {X 0,Y 199.972,Z 822.977,A -85,B 0,C 180,E1 -22598.659,E2 -22598.659} C_VEL
LIN {X 0,Y 200.595,Z 809.053,A -85,B 0,C 180,E1 -22599.457,E2 -22599.457} C_VEL
LIN {X 0,Y 201.837,Z 773.849,A -85,B 0,C 180,E1 -22600.777,E2 -22600.777} C_VEL
LIN {X 0,Y 192.608,Z 754.826,A -85,B 0,C 180,E1 -22603.358,E2 -22603.358} C_VEL
LIN {X 0,Y 184.536,Z 740.778,A -85,B 0,C 180,E1 -22605.759,E2 -22605.759} C_VEL
LIN {X 0,Y 180.345,Z 734.016,A -85,B 0,C 180,E1 -22607.081,E2 -22607.081} C_VEL
LIN {X 0,Y 178.859,Z 731.326,A -85,B 0,C 180,E1 -22607.6,E2 -22607.6} C_VEL
LIN {X 0,Y 178.616,Z 730.321,A -85,B 0,C 180,E1 -22608.128,E2 -22608.128} C_VEL
LIN {X 0,Y 178.471,Z 730.256,A -85,B 0,C 180,E1 -22613.194,E2 -22613.194} C_VEL
LIN {X 0,Y 178.429,Z 730.234,A -85,B 0,C 180,E1 -22618.211,E2 -22618.211} C_VEL
LIN {X 0,Y 178.49,Z 730.211,A -85,B 0,C 180,E1 -22623.456,E2 -22623.456} C_VEL
LIN {X 0,Y 178.394,Z 730.261,A -85,B 0,C 180,E1 -22629.079,E2 -22629.079} C_VEL
LIN {X 0,Y 178.401,Z 730.264,A -85,B 0,C 180,E1 -22632.049,E2 -22632.049} C_VEL
LIN {X 0,Y 178.458,Z 730.433,A -85,B 0,C 180,E1 -22635.348,E2 -22635.348} C_VEL
LIN {X 0,Y 178.654,Z 731.257,A -85,B 0,C 180,E1 -22635.686,E2 -22635.686} C_VEL
LIN {X 0,Y 189.005,Z 761.801,A -85,B 0,C 180,E1 -22638.459,E2 -22638.459} C_VEL
LIN {X 0,Y 186.937,Z 811.362,A -85,B 0,C 180,E1 -22641.345,E2 -22641.345} C_VEL
LIN {X 0,Y 186.319,Z 822.553,A -85,B 0,C 180,E1 -22642.273,E2 -22642.273} C_VEL
LIN {X 0,Y 185.383,Z 833.778,A -85,B 0,C 180,E1 -22643.506,E2 -22643.506} C_VEL
LIN {X 0,Y 184.522,Z 843.378,A -85,B 0,C 180,E1 -22644.824,E2 -22644.824} C_VEL
LIN {X 0,Y 183.419,Z 853.832,A -85,B 0,C 180,E1 -22646.577,E2 -22646.577} C_VEL
LIN {X 0,Y 182.439,Z 862.684,A -85,B 0,C 180,E1 -22648.359,E2 -22648.359} C_VEL
LIN {X 0,Y 181.424,Z 871.285,A -85,B 0,C 180,E1 -22650.402,E2 -22650.402} C_VEL
LIN {X 0,Y 180.451,Z 879.329,A -85,B 0,C 180,E1 -22652.646,E2 -22652.646} C_VEL
LIN {X 0,Y 179.704,Z 886.92,A -85,B 0,C 180,E1 -22655.138,E2 -22655.138} C_VEL
LIN {X 0,Y 179.154,Z 893.148,A -85,B 0,C 180,E1 -22657.512,E2 -22657.512} C_VEL
LIN {X 0,Y 178.698,Z 900.169,A -85,B 0,C 180,E1 -22660.725,E2 -22660.725} C_VEL
LIN {X 0,Y 178.583,Z 904.155,A -85,B 0,C 180,E1 -22662.833,E2 -22662.833} C_VEL
LIN {X 0,Y 178.791,Z 909.612,A -85,B 0,C 180,E1 -22666.358,E2 -22666.358} C_VEL
LIN {X 0,Y 179.492,Z 913.859,A -85,B 0,C 180,E1 -22669.851,E2 -22669.851} C_VEL
LIN {X 0,Y 180.697,Z 917.036,A -85,B 0,C 180,E1 -22673.299,E2 -22673.299} C_VEL
LIN {X 0,Y 183.177,Z 919.75,A -85,B 0,C 180,E1 -22677.801,E2 -22677.801} C_VEL
LIN {X 0,Y 184.745,Z 920.427,A -85,B 0,C 180,E1 -22680,E2 -22680} C_VEL
LIN {X 0,Y 186.554,Z 920.697,A -85,B 0,C 180,E1 -22682.159,E2 -22682.159} C_VEL
LIN {X 0,Y 190.963,Z 919.973,A -85,B 0,C 180,E1 -22686.421,E2 -22686.421} C_VEL
LIN {X 0,Y 195.999,Z 917.561,A -85,B 0,C 180,E1 -22690.328,E2 -22690.328} C_VEL
LIN {X 0,Y 198.933,Z 915.815,A -85,B 0,C 180,E1 -22692.238,E2 -22692.238} C_VEL
LIN {X 0,Y 203.738,Z 912.131,A -85,B 0,C 180,E1 -22695.003,E2 -22695.003} C_VEL
LIN {X 0,Y 208.811,Z 907.393,A -85,B 0,C 180,E1 -22697.633,E2 -22697.633} C_VEL
LIN {X 0,Y 214.329,Z 901.365,A -85,B 0,C 180,E1 -22700.139,E2 -22700.139} C_VEL
LIN {X 0,Y 220.217,Z 893.88,A -85,B 0,C 180,E1 -22702.517,E2 -22702.517} C_VEL
LIN {X 0,Y 225.396,Z 886.245,A -85,B 0,C 180,E1 -22704.439,E2 -22704.439} C_VEL
LIN {X 0,Y 230.602,Z 877.359,A -85,B 0,C 180,E1 -22706.226,E2 -22706.226} C_VEL
LIN {X 0,Y 236.038,Z 866.379,A -85,B 0,C 180,E1 -22707.966,E2 -22707.966} C_VEL
LIN {X 0,Y 240.379,Z 855.373,A -85,B 0,C 180,E1 -22709.322,E2 -22709.322} C_VEL
LIN {X 0,Y 243.608,Z 845.501,A -85,B 0,C 180,E1 -22710.322,E2 -22710.322} C_VEL
LIN {X 0,Y 246.367,Z 834.751,A -85,B 0,C 180,E1 -22711.185,E2 -22711.185} C_VEL
LIN {X 0,Y 250.181,Z 815.193,A -85,B 0,C 180,E1 -22712.345,E2 -22712.345} C_VEL
LIN {X 0,Y 250.602,Z 812.886,A -85,B 0,C 180,E1 -22712.499,E2 -22712.499} C_VEL
LIN {X 0,Y 250.246,Z 811.786,A -85,B 0,C 180,E1 -22713.447,E2 -22713.447} C_VEL
LIN {X 0,Y 249.8,Z 810.329,A -85,B 0,C 180,E1 -22715.32,E2 -22715.32} C_VEL
LIN {X 0,Y 249.532,Z 810.454,A -85,B 0,C 180,E1 -22717.062,E2 -22717.062} C_VEL
LIN {X 0,Y 249.636,Z 811.822,A -85,B 0,C 180,E1 -22719.435,E2 -22719.435} C_VEL
LIN {X 0,Y 249.683,Z 813.343,A -85,B 0,C 180,E1 -22720.41,E2 -22720.41} C_VEL
LIN {X 0,Y 249.519,Z 814.839,A -85,B 0,C 180,E1 -22720.712,E2 -22720.712} C_VEL
LIN {X 0,Y 246.762,Z 831.697,A -85,B 0,C 180,E1 -22722.38,E2 -22722.38} C_VEL
LIN {X 0,Y 245.368,Z 840.614,A -85,B 0,C 180,E1 -22723.113,E2 -22723.113} C_VEL
LIN {X 0,Y 244.07,Z 846.427,A -85,B 0,C 180,E1 -22723.324,E2 -22723.324} C_VEL
LIN {X 0,Y 240.962,Z 856.05,A -85,B 0,C 180,E1 -22723.258,E2 -22723.258} C_VEL
LIN {X 0,Y 237.331,Z 865.338,A -85,B 0,C 180,E1 -22723.182,E2 -22723.182} C_VEL
LIN {X 0,Y 235.202,Z 870.556,A -85,B 0,C 180,E1 -22723.376,E2 -22723.376} C_VEL
LIN {X 0,Y 229.002,Z 884.587,A -85,B 0,C 180,E1 -22724.474,E2 -22724.474} C_VEL
LIN {X 0,Y 223.391,Z 895.289,A -85,B 0,C 180,E1 -22725.57,E2 -22725.57} C_VEL
LIN {X 0,Y 217.341,Z 905.436,A -85,B 0,C 180,E1 -22726.91,E2 -22726.91} C_VEL
LIN {X 0,Y 211.672,Z 914.049,A -85,B 0,C 180,E1 -22728.388,E2 -22728.388} C_VEL
LIN {X 0,Y 205.656,Z 922.366,A -85,B 0,C 180,E1 -22730.148,E2 -22730.148} C_VEL
LIN {X 0,Y 198.921,Z 930.787,A -85,B 0,C 180,E1 -22732.447,E2 -22732.447} C_VEL
LIN {X 0,Y 193.805,Z 936.838,A -85,B 0,C 180,E1 -22734.531,E2 -22734.531} C_VEL
LIN {X 0,Y 188.233,Z 942.979,A -85,B 0,C 180,E1 -22737.219,E2 -22737.219} C_VEL
LIN {X 0,Y 183.355,Z 948.137,A -85,B 0,C 180,E1 -22740.11,E2 -22740.11} C_VEL
LIN {X 0,Y 179.213,Z 952.362,A -85,B 0,C 180,E1 -22743.19,E2 -22743.19} C_VEL
LIN {X 0,Y 175.872,Z 955.752,A -85,B 0,C 180,E1 -22746.443,E2 -22746.443} C_VEL
LIN {X 0,Y 172.673,Z 958.957,A -85,B 0,C 180,E1 -22750.994,E2 -22750.994} C_VEL
LIN {X 0,Y 170.933,Z 960.802,A -85,B 0,C 180,E1 -22755.715,E2 -22755.715} C_VEL
LIN {X 0,Y 170.595,Z 961.555,A -85,B 0,C 180,E1 -22759.613,E2 -22759.613} C_VEL
LIN {X 0,Y 170.576,Z 964.589,A -85,B 0,C 180,E1 -22762.896,E2 -22762.896} C_VEL
LIN {X 0,Y 170.876,Z 966.265,A -85,B 0,C 180,E1 -22765.278,E2 -22765.278} C_VEL
LIN {X 0,Y 171.172,Z 967.485,A -85,B 0,C 180,E1 -22767.643,E2 -22767.643} C_VEL
LIN {X 0,Y 171.519,Z 968.234,A -85,B 0,C 180,E1 -22769.996,E2 -22769.996} C_VEL
LIN {X 0,Y 171.097,Z 968.406,A -85,B 0,C 180,E1 -22772.351,E2 -22772.351} C_VEL
LIN {X 0,Y 170.676,Z 968.156,A -85,B 0,C 180,E1 -22774.72,E2 -22774.72} C_VEL
LIN {X 0,Y 170.266,Z 967.209,A -85,B 0,C 180,E1 -22777.847,E2 -22777.847} C_VEL
LIN {X 0,Y 170.277,Z 964.945,A -85,B 0,C 180,E1 -22781.906,E2 -22781.906} C_VEL
LIN {X 0,Y 171.464,Z 960.78,A -85,B 0,C 180,E1 -22786.67,E2 -22786.67} C_VEL
LIN {X 0,Y 173.083,Z 956.482,A -85,B 0,C 180,E1 -22790.186,E2 -22790.186} C_VEL
LIN {X 0,Y 176.26,Z 950.128,A -85,B 0,C 180,E1 -22794.119,E2 -22794.119} C_VEL
LIN {X 0,Y 179.498,Z 943.276,A -85,B 0,C 180,E1 -22797.387,E2 -22797.387} C_VEL
LIN {X 0,Y 183.646,Z 934.909,A -85,B 0,C 180,E1 -22800.465,E2 -22800.465} C_VEL
LIN {X 0,Y 187.496,Z 926.456,A -85,B 0,C 180,E1 -22802.919,E2 -22802.919} C_VEL
LIN {X 0,Y 191.913,Z 916.236,A -85,B 0,C 180,E1 -22805.22,E2 -22805.22} C_VEL
LIN {X 0,Y 196.187,Z 904.767,A -85,B 0,C 180,E1 -22807.19,E2 -22807.19} C_VEL
LIN {X 0,Y 199.691,Z 893.63,A -85,B 0,C 180,E1 -22808.656,E2 -22808.656} C_VEL
LIN {X 0,Y 202.493,Z 882.519,A -85,B 0,C 180,E1 -22809.781,E2 -22809.781} C_VEL
LIN {X 0,Y 204.928,Z 869.862,A -85,B 0,C 180,E1 -22810.717,E2 -22810.717} C_VEL
LIN {X 0,Y 206.6,Z 856.136,A -85,B 0,C 180,E1 -22811.377,E2 -22811.377} C_VEL
LIN {X 0,Y 207.345,Z 843.385,A -85,B 0,C 180,E1 -22811.862,E2 -22811.862} C_VEL
LIN {X 0,Y 206.799,Z 822.83,A -85,B 0,C 180,E1 -22813.155,E2 -22813.155} C_VEL
LIN {X 0,Y 205.925,Z 804.12,A -85,B 0,C 180,E1 -22814.495,E2 -22814.495} C_VEL
LIN {X 0,Y 205.195,Z 795.896,A -85,B 0,C 180,E1 -22815.22,E2 -22815.22} C_VEL
LIN {X 0,Y 201.937,Z 787.373,A -85,B 0,C 180,E1 -22816.914,E2 -22816.914} C_VEL
LIN {X 0,Y 198.091,Z 778.727,A -85,B 0,C 180,E1 -22819.019,E2 -22819.019} C_VEL
LIN {X 0,Y 195.113,Z 772.635,A -85,B 0,C 180,E1 -22820.758,E2 -22820.758} C_VEL
LIN {X 0,Y 192.764,Z 767.935,A -85,B 0,C 180,E1 -22822.253,E2 -22822.253} C_VEL
LIN {X 0,Y 189.339,Z 761.634,A -85,B 0,C 180,E1 -22824.588,E2 -22824.588} C_VEL
LIN {X 0,Y 185.191,Z 754.321,A -85,B 0,C 180,E1 -22827.907,E2 -22827.907} C_VEL
LIN {X 0,Y 179.91,Z 745.572,A -85,B 0,C 180,E1 -22833.264,E2 -22833.264} C_VEL
LIN {X 0,Y 175.435,Z 738.672,A -85,B 0,C 180,E1 -22840.454,E2 -22840.454} C_VEL
LIN {X 0,Y 174.199,Z 735.797,A -85,B 0,C 180,E1 -22845.186,E2 -22845.186} C_VEL
LIN {X 0,Y 173.991,Z 735.333,A -85,B 0,C 180,E1 -22850.702,E2 -22850.702} C_VEL
LIN {X 0,Y 177.653,Z 737.328,A -85,B 0,C 180,E1 -22860,E2 -22860} C_VEL
LIN {X 0,Y 179.566,Z 741.117,A -85,B 0,C 180,E1 -22862.945,E2 -22862.945} C_VEL
LIN {X 0,Y 182.278,Z 743.196,A -85,B 0,C 180,E1 -22865.809,E2 -22865.809} C_VEL
LIN {X 0,Y 184.404,Z 746.648,A -85,B 0,C 180,E1 -22867.924,E2 -22867.924} C_VEL
LIN {X 0,Y 186.268,Z 748.403,A -85,B 0,C 180,E1 -22869.437,E2 -22869.437} C_VEL
LIN {X 0,Y 188.616,Z 751.97,A -85,B 0,C 180,E1 -22871.29,E2 -22871.29} C_VEL
LIN {X 0,Y 190.215,Z 753.722,A -85,B 0,C 180,E1 -22872.402,E2 -22872.402} C_VEL
LIN {X 0,Y 192.899,Z 757.413,A -85,B 0,C 180,E1 -22874.166,E2 -22874.166} C_VEL
LIN {X 0,Y 197.538,Z 764.365,A -85,B 0,C 180,E1 -22876.928,E2 -22876.928} C_VEL
LIN {X 0,Y 202.891,Z 772.653,A -85,B 0,C 180,E1 -22879.688,E2 -22879.688} C_VEL
LIN {X 0,Y 208.15,Z 782.101,A -85,B 0,C 180,E1 -22882.152,E2 -22882.152} C_VEL
LIN {X 0,Y 211.044,Z 787.986,A -85,B 0,C 180,E1 -22883.426,E2 -22883.426} C_VEL
LIN {X 0,Y 209.394,Z 819.978,A -85,B 0,C 180,E1 -22884.72,E2 -22884.72} C_VEL
LIN {X 0,Y 208.159,Z 833.165,A -85,B 0,C 180,E1 -22885.628,E2 -22885.628} C_VEL
LIN {X 0,Y 206.056,Z 846.439,A -85,B 0,C 180,E1 -22886.92,E2 -22886.92} C_VEL
LIN {X 0,Y 203.591,Z 857.384,A -85,B 0,C 180,E1 -22888.335,E2 -22888.335} C_VEL
LIN {X 0,Y 200.35,Z 868.824,A -85,B 0,C 180,E1 -22890.26,E2 -22890.26} C_VEL
LIN {X 0,Y 196.904,Z 878.731,A -85,B 0,C 180,E1 -22892.371,E2 -22892.371} C_VEL
LIN {X 0,Y 192.95,Z 888.273,A -85,B 0,C 180,E1 -22894.969,E2 -22894.969} C_VEL
LIN {X 0,Y 189.087,Z 896.445,A -85,B 0,C 180,E1 -22897.837,E2 -22897.837} C_VEL
LIN {X 0,Y 185.577,Z 902.994,A -85,B 0,C 180,E1 -22900.768,E2 -22900.768} C_VEL
LIN {X 0,Y 182.45,Z 908.384,A -85,B 0,C 180,E1 -22903.898,E2 -22903.898} C_VEL
LIN {X 0,Y 179.84,Z 912.328,A -85,B 0,C 180,E1 -22906.857,E2 -22906.857} C_VEL
LIN {X 0,Y 177.142,Z 916.004,A -85,B 0,C 180,E1 -22910.6,E2 -22910.6} C_VEL
LIN {X 0,Y 175.733,Z 917.708,A -85,B 0,C 180,E1 -22913.143,E2 -22913.143} C_VEL
LIN {X 0,Y 174.592,Z 918.916,A -85,B 0,C 180,E1 -22915.703,E2 -22915.703} C_VEL
LIN {X 0,Y 173.684,Z 919.62,A -85,B 0,C 180,E1 -22918.266,E2 -22918.266} C_VEL
LIN {X 0,Y 173.019,Z 919.828,A -85,B 0,C 180,E1 -22920.832,E2 -22920.832} C_VEL
LIN {X 0,Y 172.595,Z 919.552,A -85,B 0,C 180,E1 -22923.617,E2 -22923.617} C_VEL
LIN {X 0,Y 172.47,Z 918.854,A -85,B 0,C 180,E1 -22925.957,E2 -22925.957} C_VEL
LIN {X 0,Y 172.63,Z 917.112,A -85,B 0,C 180,E1 -22929.451,E2 -22929.451} C_VEL
LIN {X 0,Y 173.469,Z 913.867,A -85,B 0,C 180,E1 -22933.528,E2 -22933.528} C_VEL
LIN {X 0,Y 174.755,Z 909.707,A -85,B 0,C 180,E1 -22937.225,E2 -22937.225} C_VEL
LIN {X 0,Y 176.453,Z 904.341,A -85,B 0,C 180,E1 -22940.836,E2 -22940.836} C_VEL
LIN {X 0,Y 178.651,Z 897.573,A -85,B 0,C 180,E1 -22944.359,E2 -22944.359} C_VEL
LIN {X 0,Y 181.267,Z 889.098,A -85,B 0,C 180,E1 -22947.781,E2 -22947.781} C_VEL
LIN {X 0,Y 183.723,Z 880.483,A -85,B 0,C 180,E1 -22950.551,E2 -22950.551} C_VEL
LIN {X 0,Y 186.214,Z 871.065,A -85,B 0,C 180,E1 -22952.978,E2 -22952.978} C_VEL
LIN {X 0,Y 188.484,Z 860.875,A -85,B 0,C 180,E1 -22955.084,E2 -22955.084} C_VEL
LIN {X 0,Y 190.874,Z 848.591,A -85,B 0,C 180,E1 -22957.048,E2 -22957.048} C_VEL
LIN {X 0,Y 192.664,Z 836.376,A -85,B 0,C 180,E1 -22958.538,E2 -22958.538} C_VEL
LIN {X 0,Y 193.849,Z 823.37,A -85,B 0,C 180,E1 -22959.69,E2 -22959.69} C_VEL
LIN {X 0,Y 194.493,Z 810.15,A -85,B 0,C 180,E1 -22960.458,E2 -22960.458} C_VEL
LIN {X 0,Y 195.678,Z 776.027,A -85,B 0,C 180,E1 -22961.79,E2 -22961.79} C_VEL
LIN {X 0,Y 187.357,Z 758.501,A -85,B 0,C 180,E1 -22964.265,E2 -22964.265} C_VEL
LIN {X 0,Y 178.191,Z 742.661,A -85,B 0,C 180,E1 -22967.145,E2 -22967.145} C_VEL
LIN {X 0,Y 173.51,Z 735.171,A -85,B 0,C 180,E1 -22968.717,E2 -22968.717} C_VEL
LIN {X 0,Y 171.846,Z 732.529,A -85,B 0,C 180,E1 -22969.322,E2 -22969.322} C_VEL
LIN {X 0,Y 171.515,Z 731.386,A -85,B 0,C 180,E1 -22969.74,E2 -22969.74} C_VEL
LIN {X 0,Y 171.422,Z 731.116,A -85,B 0,C 180,E1 -22971.657,E2 -22971.657} C_VEL
LIN {X 0,Y 171.367,Z 731.105,A -85,B 0,C 180,E1 -22976.82,E2 -22976.82} C_VEL
LIN {X 0,Y 171.412,Z 731.135,A -85,B 0,C 180,E1 -22980.568,E2 -22980.568} C_VEL
LIN {X 0,Y 171.399,Z 731.087,A -85,B 0,C 180,E1 -22985.037,E2 -22985.037} C_VEL
LIN {X 0,Y 171.35,Z 731.136,A -85,B 0,C 180,E1 -22988.803,E2 -22988.803} C_VEL
LIN {X 0,Y 171.401,Z 731.228,A -85,B 0,C 180,E1 -22994.659,E2 -22994.659} C_VEL
LIN {X 0,Y 171.552,Z 732.034,A -85,B 0,C 180,E1 -22995.075,E2 -22995.075} C_VEL
LIN {X 0,Y 182.092,Z 763.115,A -85,B 0,C 180,E1 -22998.027,E2 -22998.027} C_VEL
LIN {X 0,Y 179.842,Z 813.233,A -85,B 0,C 180,E1 -23001.118,E2 -23001.118} C_VEL
LIN {X 0,Y 179.236,Z 823.704,A -85,B 0,C 180,E1 -23002.039,E2 -23002.039} C_VEL
LIN {X 0,Y 178.32,Z 834.238,A -85,B 0,C 180,E1 -23003.232,E2 -23003.232} C_VEL
LIN {X 0,Y 177.437,Z 843.944,A -85,B 0,C 180,E1 -23004.6,E2 -23004.6} C_VEL
LIN {X 0,Y 176.334,Z 854.376,A -85,B 0,C 180,E1 -23006.4,E2 -23006.4} C_VEL
LIN {X 0,Y 175.286,Z 863.64,A -85,B 0,C 180,E1 -23008.325,E2 -23008.325} C_VEL
LIN {X 0,Y 174.263,Z 872.074,A -85,B 0,C 180,E1 -23010.393,E2 -23010.393} C_VEL
LIN {X 0,Y 173.247,Z 880.754,A -85,B 0,C 180,E1 -23012.912,E2 -23012.912} C_VEL
LIN {X 0,Y 172.541,Z 887.783,A -85,B 0,C 180,E1 -23015.322,E2 -23015.322} C_VEL
LIN {X 0,Y 171.898,Z 895.364,A -85,B 0,C 180,E1 -23018.409,E2 -23018.409} C_VEL
LIN {X 0,Y 171.559,Z 901.694,A -85,B 0,C 180,E1 -23021.489,E2 -23021.489} C_VEL
LIN {X 0,Y 171.514,Z 906.977,A -85,B 0,C 180,E1 -23024.553,E2 -23024.553} C_VEL
LIN {X 0,Y 171.777,Z 910.631,A -85,B 0,C 180,E1 -23026.995,E2 -23026.995} C_VEL
LIN {X 0,Y 172.626,Z 914.944,A -85,B 0,C 180,E1 -23030.627,E2 -23030.627} C_VEL
LIN {X 0,Y 173.438,Z 917.17,A -85,B 0,C 180,E1 -23033.017,E2 -23033.017} C_VEL
LIN {X 0,Y 175.958,Z 920.427,A -85,B 0,C 180,E1 -23037.711,E2 -23037.711} C_VEL
LIN {X 0,Y 177.53,Z 921.382,A -85,B 0,C 180,E1 -23040,E2 -23040} C_VEL
LIN {X 0,Y 179.4,Z 921.935,A -85,B 0,C 180,E1 -23042.245,E2 -23042.245} C_VEL
LIN {X 0,Y 181.49,Z 922.07,A -85,B 0,C 180,E1 -23044.442,E2 -23044.442} C_VEL
LIN {X 0,Y 186.381,Z 920.999,A -85,B 0,C 180,E1 -23048.675,E2 -23048.675} C_VEL
LIN {X 0,Y 189.167,Z 919.981,A -85,B 0,C 180,E1 -23050.705,E2 -23050.705} C_VEL
LIN {X 0,Y 193.769,Z 917.487,A -85,B 0,C 180,E1 -23053.636,E2 -23053.636} C_VEL
LIN {X 0,Y 198.887,Z 913.966,A -85,B 0,C 180,E1 -23056.421,E2 -23056.421} C_VEL
LIN {X 0,Y 204.288,Z 909.369,A -85,B 0,C 180,E1 -23059.076,E2 -23059.076} C_VEL
LIN {X 0,Y 210.145,Z 903.508,A -85,B 0,C 180,E1 -23061.585,E2 -23061.585} C_VEL
LIN {X 0,Y 215.374,Z 897.48,A -85,B 0,C 180,E1 -23063.591,E2 -23063.591} C_VEL
LIN {X 0,Y 220.815,Z 890.254,A -85,B 0,C 180,E1 -23065.525,E2 -23065.525} C_VEL
LIN {X 0,Y 226.174,Z 882.024,A -85,B 0,C 180,E1 -23067.279,E2 -23067.279} C_VEL
LIN {X 0,Y 231.242,Z 872.943,A -85,B 0,C 180,E1 -23068.847,E2 -23068.847} C_VEL
LIN {X 0,Y 235.54,Z 863.99,A -85,B 0,C 180,E1 -23070.079,E2 -23070.079} C_VEL
LIN {X 0,Y 239.297,Z 854.542,A -85,B 0,C 180,E1 -23071.174,E2 -23071.174} C_VEL
LIN {X 0,Y 242.704,Z 844.24,A -85,B 0,C 180,E1 -23072.146,E2 -23072.146} C_VEL
LIN {X 0,Y 245.928,Z 831.62,A -85,B 0,C 180,E1 -23073.062,E2 -23073.062} C_VEL
LIN {X 0,Y 248.496,Z 818.491,A -85,B 0,C 180,E1 -23073.829,E2 -23073.829} C_VEL
LIN {X 0,Y 248.164,Z 817.196,A -85,B 0,C 180,E1 -23075.588,E2 -23075.588} C_VEL
LIN {X 0,Y 247.936,Z 817.489,A -85,B 0,C 180,E1 -23077.215,E2 -23077.215} C_VEL
LIN {X 0,Y 247.986,Z 818.696,A -85,B 0,C 180,E1 -23079.17,E2 -23079.17} C_VEL
LIN {X 0,Y 247.958,Z 819.167,A -85,B 0,C 180,E1 -23079.411,E2 -23079.411} C_VEL
LIN {X 0,Y 244.667,Z 837.18,A -85,B 0,C 180,E1 -23081.129,E2 -23081.129} C_VEL
LIN {X 0,Y 241.416,Z 852.022,A -85,B 0,C 180,E1 -23082.282,E2 -23082.282} C_VEL
LIN {X 0,Y 236.898,Z 866.031,A -85,B 0,C 180,E1 -23083.098,E2 -23083.098} C_VEL
LIN {X 0,Y 235.202,Z 870.556,A -85,B 0,C 180,E1 -23083.376,E2 -23083.376} C_VEL
LIN {X 0,Y 232.853,Z 875.924,A -85,B 0,C 180,E1 -23083.594,E2 -23083.594} C_VEL
LIN {X 0,Y 227.907,Z 884.55,A -85,B 0,C 180,E1 -23083.619,E2 -23083.619} C_VEL
LIN {X 0,Y 222.514,Z 892.95,A -85,B 0,C 180,E1 -23083.733,E2 -23083.733} C_VEL
LIN {X 0,Y 219.45,Z 897.59,A -85,B 0,C 180,E1 -23084.1,E2 -23084.1} C_VEL
LIN {X 0,Y 211.679,Z 909.442,A -85,B 0,C 180,E1 -23085.792,E2 -23085.792} C_VEL
LIN {X 0,Y 204.012,Z 919.633,A -85,B 0,C 180,E1 -23087.794,E2 -23087.794} C_VEL
LIN {X 0,Y 196.835,Z 928.177,A -85,B 0,C 180,E1 -23090.004,E2 -23090.004} C_VEL
LIN {X 0,Y 191.213,Z 934.356,A -85,B 0,C 180,E1 -23091.998,E2 -23091.998} C_VEL
LIN {X 0,Y 184.158,Z 941.517,A -85,B 0,C 180,E1 -23095.075,E2 -23095.075} C_VEL
LIN {X 0,Y 178.85,Z 946.618,A -85,B 0,C 180,E1 -23097.958,E2 -23097.958} C_VEL
LIN {X 0,Y 174.252,Z 950.828,A -85,B 0,C 180,E1 -23101.05,E2 -23101.05} C_VEL
LIN {X 0,Y 169.348,Z 955.054,A -85,B 0,C 180,E1 -23105.477,E2 -23105.477} C_VEL
LIN {X 0,Y 167.387,Z 956.724,A -85,B 0,C 180,E1 -23107.794,E2 -23107.794} C_VEL
LIN {X 0,Y 164.754,Z 958.974,A -85,B 0,C 180,E1 -23112.623,E2 -23112.623} C_VEL
LIN {X 0,Y 163.674,Z 959.818,A -85,B 0,C 180,E1 -23117.599,E2 -23117.599} C_VEL
LIN {X 0,Y 163.635,Z 959.974,A -85,B 0,C 180,E1 -23118.853,E2 -23118.853} C_VEL
LIN {X 0,Y 163.513,Z 963.397,A -85,B 0,C 180,E1 -23122.588,E2 -23122.588} C_VEL
LIN {X 0,Y 163.786,Z 965.106,A -85,B 0,C 180,E1 -23125.073,E2 -23125.073} C_VEL
LIN {X 0,Y 164.109,Z 966.362,A -85,B 0,C 180,E1 -23127.542,E2 -23127.542} C_VEL
LIN {X 0,Y 164.475,Z 967.169,A -85,B 0,C 180,E1 -23129.996,E2 -23129.996} C_VEL
LIN {X 0,Y 164.024,Z 967.369,A -85,B 0,C 180,E1 -23132.452,E2 -23132.452} C_VEL
LIN {X 0,Y 163.586,Z 967.143,A -85,B 0,C 180,E1 -23134.925,E2 -23134.925} C_VEL
LIN {X 0,Y 163.199,Z 966.353,A -85,B 0,C 180,E1 -23137.916,E2 -23137.916} C_VEL
LIN {X 0,Y 163.278,Z 964.047,A -85,B 0,C 180,E1 -23142.424,E2 -23142.424} C_VEL
LIN {X 0,Y 164.587,Z 959.942,A -85,B 0,C 180,E1 -23147.388,E2 -23147.388} C_VEL
LIN {X 0,Y 166.375,Z 955.729,A -85,B 0,C 180,E1 -23151.038,E2 -23151.038} C_VEL
LIN {X 0,Y 169.743,Z 949.504,A -85,B 0,C 180,E1 -23155.108,E2 -23155.108} C_VEL
LIN {X 0,Y 173.201,Z 942.759,A -85,B 0,C 180,E1 -23158.471,E2 -23158.471} C_VEL
LIN {X 0,Y 177.539,Z 934.497,A -85,B 0,C 180,E1 -23161.631,E2 -23161.631} C_VEL
LIN {X 0,Y 181.582,Z 926.17,A -85,B 0,C 180,E1 -23164.135,E2 -23164.135} C_VEL
LIN {X 0,Y 186.167,Z 916.115,A -85,B 0,C 180,E1 -23166.478,E2 -23166.478} C_VEL
LIN {X 0,Y 190.586,Z 904.964,A -85,B 0,C 180,E1 -23168.478,E2 -23168.478} C_VEL
LIN {X 0,Y 194.209,Z 894.156,A -85,B 0,C 180,E1 -23169.962,E2 -23169.962} C_VEL
LIN {X 0,Y 197.113,Z 883.517,A -85,B 0,C 180,E1 -23171.096,E2 -23171.096} C_VEL
LIN {X 0,Y 199.921,Z 870.185,A -85,B 0,C 180,E1 -23172.132,E2 -23172.132} C_VEL
LIN {X 0,Y 201.759,Z 856.706,A -85,B 0,C 180,E1 -23172.827,E2 -23172.827} C_VEL
LIN {X 0,Y 202.58,Z 844.243,A -85,B 0,C 180,E1 -23173.308,E2 -23173.308} C_VEL
LIN {X 0,Y 202.156,Z 824.372,A -85,B 0,C 180,E1 -23174.595,E2 -23174.595} C_VEL
LIN {X 0,Y 201.373,Z 805.003,A -85,B 0,C 180,E1 -23176.029,E2 -23176.029} C_VEL
LIN {X 0,Y 200.83,Z 798.822,A -85,B 0,C 180,E1 -23176.616,E2 -23176.616} C_VEL
LIN {X 0,Y 197.536,Z 790.1,A -85,B 0,C 180,E1 -23178.486,E2 -23178.486} C_VEL
LIN {X 0,Y 193.269,Z 780.251,A -85,B 0,C 180,E1 -23181.068,E2 -23181.068} C_VEL
LIN {X 0,Y 190.043,Z 773.685,A -85,B 0,C 180,E1 -23183.205,E2 -23183.205} C_VEL
LIN {X 0,Y 186.826,Z 767.477,A -85,B 0,C 180,E1 -23185.57,E2 -23185.57} C_VEL
LIN {X 0,Y 183.068,Z 760.523,A -85,B 0,C 180,E1 -23188.769,E2 -23188.769} C_VEL
LIN {X 0,Y 178.301,Z 752.132,A -85,B 0,C 180,E1 -23193.978,E2 -23193.978} C_VEL
LIN {X 0,Y 174.299,Z 745.55,A -85,B 0,C 180,E1 -23200.896,E2 -23200.896} C_VEL
LIN {X 0,Y 173.214,Z 742.816,A -85,B 0,C 180,E1 -23205.31,E2 -23205.31} C_VEL
LIN {X 0,Y 173.044,Z 742.371,A -85,B 0,C 180,E1 -23210.651,E2 -23210.651} C_VEL
LIN {X 0,Y 176.387,Z 744.29,A -85,B 0,C 180,E1 -23219.572,E2 -23219.572} C_VEL
LIN {X 0,Y 178.043,Z 747.716,A -85,B 0,C 180,E1 -23222.263,E2 -23222.263} C_VEL
LIN {X 0,Y 180.665,Z 750.006,A -85,B 0,C 180,E1 -23225.232,E2 -23225.232} C_VEL
LIN {X 0,Y 182.851,Z 753.436,A -85,B 0,C 180,E1 -23227.476,E2 -23227.476} C_VEL
LIN {X 0,Y 184.411,Z 755.16,A -85,B 0,C 180,E1 -23228.838,E2 -23228.838} C_VEL
LIN {X 0,Y 186.885,Z 758.741,A -85,B 0,C 180,E1 -23230.838,E2 -23230.838} C_VEL
LIN {X 0,Y 187.977,Z 760.051,A -85,B 0,C 180,E1 -23231.636,E2 -23231.636} C_VEL
LIN {X 0,Y 191.38,Z 765.063,A -85,B 0,C 180,E1 -23233.987,E2 -23233.987} C_VEL
LIN {X 0,Y 195.915,Z 771.941,A -85,B 0,C 180,E1 -23236.734,E2 -23236.734} C_VEL
LIN {X 0,Y 201.491,Z 781.358,A -85,B 0,C 180,E1 -23239.7,E2 -23239.7} C_VEL
LIN {X 0,Y 206.256,Z 790.74,A -85,B 0,C 180,E1 -23242.013,E2 -23242.013} C_VEL
LIN {X 0,Y 204.647,Z 821.519,A -85,B 0,C 180,E1 -23243.32,E2 -23243.32} C_VEL
LIN {X 0,Y 203.293,Z 834.667,A -85,B 0,C 180,E1 -23244.245,E2 -23244.245} C_VEL
LIN {X 0,Y 201.308,Z 846.546,A -85,B 0,C 180,E1 -23245.407,E2 -23245.407} C_VEL
LIN {X 0,Y 198.811,Z 857.458,A -85,B 0,C 180,E1 -23246.807,E2 -23246.807} C_VEL
LIN {X 0,Y 195.843,Z 867.606,A -85,B 0,C 180,E1 -23248.463,E2 -23248.463} C_VEL
LIN {X 0,Y 192.155,Z 877.968,A -85,B 0,C 180,E1 -23250.617,E2 -23250.617} C_VEL
LIN {X 0,Y 188.442,Z 886.863,A -85,B 0,C 180,E1 -23252.957,E2 -23252.957} C_VEL
LIN {X 0,Y 184.233,Z 895.652,A -85,B 0,C 180,E1 -23255.899,E2 -23255.899} C_VEL
LIN {X 0,Y 180.447,Z 902.476,A -85,B 0,C 180,E1 -23258.841,E2 -23258.841} C_VEL
LIN {X 0,Y 176.425,Z 909.086,A -85,B 0,C 180,E1 -23262.627,E2 -23262.627} C_VEL
LIN {X 0,Y 173.066,Z 913.885,A -85,B 0,C 180,E1 -23266.347,E2 -23266.347} C_VEL
LIN {X 0,Y 171.106,Z 916.334,A -85,B 0,C 180,E1 -23268.92,E2 -23268.92} C_VEL
LIN {X 0,Y 169.18,Z 918.587,A -85,B 0,C 180,E1 -23272.12,E2 -23272.12} C_VEL
LIN {X 0,Y 167.095,Z 920.467,A -85,B 0,C 180,E1 -23276.858,E2 -23276.858} C_VEL
LIN {X 0,Y 166.3,Z 920.855,A -85,B 0,C 180,E1 -23279.532,E2 -23279.532} C_VEL
LIN {X 0,Y 165.623,Z 920.634,A -85,B 0,C 180,E1 -23283.014,E2 -23283.014} C_VEL
LIN {X 0,Y 165.458,Z 919.145,A -85,B 0,C 180,E1 -23287.529,E2 -23287.529} C_VEL
LIN {X 0,Y 165.681,Z 917.639,A -85,B 0,C 180,E1 -23290.167,E2 -23290.167} C_VEL
LIN {X 0,Y 166.58,Z 914.476,A -85,B 0,C 180,E1 -23294.087,E2 -23294.087} C_VEL
LIN {X 0,Y 167.936,Z 910.196,A -85,B 0,C 180,E1 -23297.926,E2 -23297.926} C_VEL
LIN {X 0,Y 169.704,Z 904.841,A -85,B 0,C 180,E1 -23301.579,E2 -23301.579} C_VEL
LIN {X 0,Y 172.092,Z 897.706,A -85,B 0,C 180,E1 -23305.319,E2 -23305.319} C_VEL
LIN {X 0,Y 174.442,Z 890.459,A -85,B 0,C 180,E1 -23308.33,E2 -23308.33} C_VEL
LIN {X 0,Y 176.968,Z 882.081,A -85,B 0,C 180,E1 -23311.141,E2 -23311.141} C_VEL
LIN {X 0,Y 179.827,Z 871.66,A -85,B 0,C 180,E1 -23313.925,E2 -23313.925} C_VEL
LIN {X 0,Y 182.199,Z 861.376,A -85,B 0,C 180,E1 -23316.092,E2 -23316.092} C_VEL
LIN {X 0,Y 184.722,Z 848.937,A -85,B 0,C 180,E1 -23318.113,E2 -23318.113} C_VEL
LIN {X 0,Y 186.452,Z 837.528,A -85,B 0,C 180,E1 -23319.533,E2 -23319.533} C_VEL
LIN {X 0,Y 187.731,Z 824.34,A -85,B 0,C 180,E1 -23320.735,E2 -23320.735} C_VEL
LIN {X 0,Y 188.399,Z 811.64,A -85,B 0,C 180,E1 -23321.501,E2 -23321.501} C_VEL
LIN {X 0,Y 189.619,Z 778.178,A -85,B 0,C 180,E1 -23322.852,E2 -23322.852} C_VEL
LIN {X 0,Y 182.326,Z 762.605,A -85,B 0,C 180,E1 -23325.151,E2 -23325.151} C_VEL
LIN {X 0,Y 173.557,Z 747.287,A -85,B 0,C 180,E1 -23328.046,E2 -23328.046} C_VEL
LIN {X 0,Y 168.895,Z 739.854,A -85,B 0,C 180,E1 -23329.696,E2 -23329.696} C_VEL
LIN {X 0,Y 166.554,Z 736.25,A -85,B 0,C 180,E1 -23330.568,E2 -23330.568} C_VEL
LIN {X 0,Y 164.884,Z 733.869,A -85,B 0,C 180,E1 -23331.209,E2 -23331.209} C_VEL
LIN {X 0,Y 164.452,Z 732.434,A -85,B 0,C 180,E1 -23331.634,E2 -23331.634} C_VEL
LIN {X 0,Y 164.341,Z 732.01,A -85,B 0,C 180,E1 -23332.64,E2 -23332.64} C_VEL
LIN {X 0,Y 164.342,Z 731.98,A -85,B 0,C 180,E1 -23336.095,E2 -23336.095} C_VEL
LIN {X 0,Y 164.351,Z 732.006,A -85,B 0,C 180,E1 -23341.212,E2 -23341.212} C_VEL
LIN {X 0,Y 164.287,Z 731.983,A -85,B 0,C 180,E1 -23346.796,E2 -23346.796} C_VEL
LIN {X 0,Y 164.293,Z 732.021,A -85,B 0,C 180,E1 -23349.92,E2 -23349.92} C_VEL
LIN {X 0,Y 164.329,Z 732.194,A -85,B 0,C 180,E1 -23354.135,E2 -23354.135} C_VEL
LIN {X 0,Y 164.52,Z 732.994,A -85,B 0,C 180,E1 -23354.498,E2 -23354.498} C_VEL
LIN {X 0,Y 175.07,Z 764.263,A -85,B 0,C 180,E1 -23357.593,E2 -23357.593} C_VEL
LIN {X 0,Y 172.845,Z 813.833,A -85,B 0,C 180,E1 -23360.781,E2 -23360.781} C_VEL
LIN {X 0,Y 172.125,Z 824.76,A -85,B 0,C 180,E1 -23361.773,E2 -23361.773} C_VEL
LIN {X 0,Y 171.169,Z 835.869,A -85,B 0,C 180,E1 -23363.095,E2 -23363.095} C_VEL
LIN {X 0,Y 170.154,Z 846.396,A -85,B 0,C 180,E1 -23364.671,E2 -23364.671} C_VEL
LIN {X 0,Y 169.263,Z 854.621,A -85,B 0,C 180,E1 -23366.148,E2 -23366.148} C_VEL
LIN {X 0,Y 168.203,Z 863.989,A -85,B 0,C 180,E1 -23368.162,E2 -23368.162} C_VEL
LIN {X 0,Y 166.984,Z 873.834,A -85,B 0,C 180,E1 -23370.707,E2 -23370.707} C_VEL
LIN {X 0,Y 165.999,Z 882.099,A -85,B 0,C 180,E1 -23373.247,E2 -23373.247} C_VEL
LIN {X 0,Y 165.398,Z 888.513,A -85,B 0,C 180,E1 -23375.525,E2 -23375.525} C_VEL
LIN {X 0,Y 164.734,Z 896.165,A -85,B 0,C 180,E1 -23378.739,E2 -23378.739} C_VEL
LIN {X 0,Y 164.42,Z 902.58,A -85,B 0,C 180,E1 -23381.947,E2 -23381.947} C_VEL
LIN {X 0,Y 164.457,Z 907.914,A -85,B 0,C 180,E1 -23385.143,E2 -23385.143} C_VEL
LIN {X 0,Y 164.958,Z 912.569,A -85,B 0,C 180,E1 -23388.512,E2 -23388.512} C_VEL
LIN {X 0,Y 165.773,Z 915.981,A -85,B 0,C 180,E1 -23391.466,E2 -23391.466} C_VEL
LIN {X 0,Y 167.349,Z 919.303,A -85,B 0,C 180,E1 -23395.181,E2 -23395.181} C_VEL
LIN {X 0,Y 170.312,Z 922.174,A -85,B 0,C 180,E1 -23400,E2 -23400} C_VEL
LIN {X 0,Y 172.222,Z 923.004,A -85,B 0,C 180,E1 -23402.338,E2 -23402.338} C_VEL
LIN {X 0,Y 174.36,Z 923.382,A -85,B 0,C 180,E1 -23404.624,E2 -23404.624} C_VEL
LIN {X 0,Y 179.427,Z 922.958,A -85,B 0,C 180,E1 -23409.014,E2 -23409.014} C_VEL
LIN {X 0,Y 185.393,Z 920.825,A -85,B 0,C 180,E1 -23413.147,E2 -23413.147} C_VEL
LIN {X 0,Y 189.801,Z 918.596,A -85,B 0,C 180,E1 -23415.681,E2 -23415.681} C_VEL
LIN {X 0,Y 196.04,Z 914.391,A -85,B 0,C 180,E1 -23418.823,E2 -23418.823} C_VEL
LIN {X 0,Y 199.95,Z 911.392,A -85,B 0,C 180,E1 -23420.578,E2 -23420.578} C_VEL
LIN {X 0,Y 206.501,Z 905.314,A -85,B 0,C 180,E1 -23423.226,E2 -23423.226} C_VEL
LIN {X 0,Y 212.671,Z 898.658,A -85,B 0,C 180,E1 -23425.442,E2 -23425.442} C_VEL
LIN {X 0,Y 218.339,Z 891.513,A -85,B 0,C 180,E1 -23427.302,E2 -23427.302} C_VEL
LIN {X 0,Y 223.016,Z 884.926,A -85,B 0,C 180,E1 -23428.723,E2 -23428.723} C_VEL
LIN {X 0,Y 228.267,Z 876.256,A -85,B 0,C 180,E1 -23430.249,E2 -23430.249} C_VEL
LIN {X 0,Y 233.209,Z 866.75,A -85,B 0,C 180,E1 -23431.575,E2 -23431.575} C_VEL
LIN {X 0,Y 237.401,Z 857.09,A -85,B 0,C 180,E1 -23432.702,E2 -23432.702} C_VEL
LIN {X 0,Y 240.437,Z 848.643,A -85,B 0,C 180,E1 -23433.509,E2 -23433.509} C_VEL
LIN {X 0,Y 243.674,Z 837.539,A -85,B 0,C 180,E1 -23434.382,E2 -23434.382} C_VEL
LIN {X 0,Y 246.622,Z 824.519,A -85,B 0,C 180,E1 -23435.169,E2 -23435.169} C_VEL
LIN {X 0,Y 246.551,Z 824.11,A -85,B 0,C 180,E1 -23435.746,E2 -23435.746} C_VEL
LIN {X 0,Y 246.312,Z 824.735,A -85,B 0,C 180,E1 -23437.841,E2 -23437.841} C_VEL
LIN {X 0,Y 246.311,Z 824.892,A -85,B 0,C 180,E1 -23438.22,E2 -23438.22} C_VEL
LIN {X 0,Y 242.864,Z 841.369,A -85,B 0,C 180,E1 -23439.758,E2 -23439.758} C_VEL
LIN {X 0,Y 239.11,Z 855.367,A -85,B 0,C 180,E1 -23440.817,E2 -23440.817} C_VEL
LIN {X 0,Y 234.63,Z 867.733,A -85,B 0,C 180,E1 -23441.507,E2 -23441.507} C_VEL
LIN {X 0,Y 228.599,Z 881.183,A -85,B 0,C 180,E1 -23442.448,E2 -23442.448} C_VEL
LIN {X 0,Y 222.023,Z 893.321,A -85,B 0,C 180,E1 -23443.603,E2 -23443.603} C_VEL
LIN {X 0,Y 219.45,Z 897.59,A -85,B 0,C 180,E1 -23444.1,E2 -23444.1} C_VEL
LIN {X 0,Y 217.211,Z 900.85,A -85,B 0,C 180,E1 -23444.325,E2 -23444.325} C_VEL
LIN {X 0,Y 208.007,Z 910.785,A -85,B 0,C 180,E1 -23444.38,E2 -23444.38} C_VEL
LIN {X 0,Y 205.548,Z 913.56,A -85,B 0,C 180,E1 -23444.72,E2 -23444.72} C_VEL
LIN {X 0,Y 196.374,Z 924.436,A -85,B 0,C 180,E1 -23447.154,E2 -23447.154} C_VEL
LIN {X 0,Y 187.964,Z 933.042,A -85,B 0,C 180,E1 -23449.832,E2 -23449.832} C_VEL
LIN {X 0,Y 182.49,Z 938.346,A -85,B 0,C 180,E1 -23451.958,E2 -23451.958} C_VEL
LIN {X 0,Y 174.646,Z 945.161,A -85,B 0,C 180,E1 -23455.706,E2 -23455.706} C_VEL
LIN {X 0,Y 169.594,Z 949.333,A -85,B 0,C 180,E1 -23458.798,E2 -23458.798} C_VEL
LIN {X 0,Y 165.289,Z 952.681,A -85,B 0,C 180,E1 -23462.11,E2 -23462.11} C_VEL
LIN {X 0,Y 160.81,Z 955.879,A -85,B 0,C 180,E1 -23466.834,E2 -23466.834} C_VEL
LIN {X 0,Y 157.984,Z 957.78,A -85,B 0,C 180,E1 -23471.853,E2 -23471.853} C_VEL
LIN {X 0,Y 156.793,Z 958.341,A -85,B 0,C 180,E1 -23477.045,E2 -23477.045} C_VEL
LIN {X 0,Y 156.685,Z 958.526,A -85,B 0,C 180,E1 -23478.187,E2 -23478.187} C_VEL
LIN {X 0,Y 156.457,Z 962.199,A -85,B 0,C 180,E1 -23482.252,E2 -23482.252} C_VEL
LIN {X 0,Y 156.701,Z 963.942,A -85,B 0,C 180,E1 -23484.85,E2 -23484.85} C_VEL
LIN {X 0,Y 157.041,Z 965.234,A -85,B 0,C 180,E1 -23487.431,E2 -23487.431} C_VEL
LIN {X 0,Y 157.43,Z 966.084,A -85,B 0,C 180,E1 -23489.996,E2 -23489.996} C_VEL
LIN {X 0,Y 156.947,Z 966.332,A -85,B 0,C 180,E1 -23492.563,E2 -23492.563} C_VEL
LIN {X 0,Y 156.505,Z 966.131,A -85,B 0,C 180,E1 -23495.149,E2 -23495.149} C_VEL
LIN {X 0,Y 156.154,Z 965.437,A -85,B 0,C 180,E1 -23498.048,E2 -23498.048} C_VEL
LIN {X 0,Y 156.287,Z 963.152,A -85,B 0,C 180,E1 -23502.99,E2 -23502.99} C_VEL
LIN {X 0,Y 157.751,Z 959.129,A -85,B 0,C 180,E1 -23508.167,E2 -23508.167} C_VEL
LIN {X 0,Y 159.727,Z 954.994,A -85,B 0,C 180,E1 -23511.958,E2 -23511.958} C_VEL
LIN {X 0,Y 162.766,Z 949.818,A -85,B 0,C 180,E1 -23515.577,E2 -23515.577} C_VEL
LIN {X 0,Y 166.973,Z 942.227,A -85,B 0,C 180,E1 -23519.637,E2 -23519.637} C_VEL
LIN {X 0,Y 171.498,Z 934.11,A -85,B 0,C 180,E1 -23522.883,E2 -23522.883} C_VEL
LIN {X 0,Y 175.758,Z 925.941,A -85,B 0,C 180,E1 -23525.432,E2 -23525.432} C_VEL
LIN {X 0,Y 180.518,Z 916.078,A -85,B 0,C 180,E1 -23527.816,E2 -23527.816} C_VEL
LIN {X 0,Y 185.09,Z 905.214,A -85,B 0,C 180,E1 -23529.844,E2 -23529.844} C_VEL
LIN {X 0,Y 188.836,Z 894.759,A -85,B 0,C 180,E1 -23531.342,E2 -23531.342} C_VEL
LIN {X 0,Y 192.139,Z 883.469,A -85,B 0,C 180,E1 -23532.581,E2 -23532.581} C_VEL
LIN {X 0,Y 195.131,Z 869.96,A -85,B 0,C 180,E1 -23533.659,E2 -23533.659} C_VEL
LIN {X 0,Y 197.083,Z 856.985,A -85,B 0,C 180,E1 -23534.354,E2 -23534.354} C_VEL
LIN {X 0,Y 197.939,Z 845.245,A -85,B 0,C 180,E1 -23534.819,E2 -23534.819} C_VEL
LIN {X 0,Y 197.611,Z 821.473,A -85,B 0,C 180,E1 -23536.413,E2 -23536.413} C_VEL
LIN {X 0,Y 196.898,Z 803.857,A -85,B 0,C 180,E1 -23537.832,E2 -23537.832} C_VEL
LIN {X 0,Y 196.587,Z 801.745,A -85,B 0,C 180,E1 -23538.099,E2 -23538.099} C_VEL
LIN {X 0,Y 193.123,Z 792.655,A -85,B 0,C 180,E1 -23540.22,E2 -23540.22} C_VEL
LIN {X 0,Y 189.662,Z 784.404,A -85,B 0,C 180,E1 -23542.544,E2 -23542.544} C_VEL
LIN {X 0,Y 187.106,Z 778.936,A -85,B 0,C 180,E1 -23544.377,E2 -23544.377} C_VEL
LIN {X 0,Y 184.373,Z 773.301,A -85,B 0,C 180,E1 -23546.577,E2 -23546.577} C_VEL
LIN {X 0,Y 180.976,Z 766.69,A -85,B 0,C 180,E1 -23549.679,E2 -23549.679} C_VEL
LIN {X 0,Y 176.605,Z 758.521,A -85,B 0,C 180,E1 -23554.865,E2 -23554.865} C_VEL
LIN {X 0,Y 173.192,Z 752.467,A -85,B 0,C 180,E1 -23561.287,E2 -23561.287} C_VEL
LIN {X 0,Y 172.165,Z 749.767,A -85,B 0,C 180,E1 -23565.823,E2 -23565.823} C_VEL
LIN {X 0,Y 172.098,Z 749.399,A -85,B 0,C 180,E1 -23570.599,E2 -23570.599} C_VEL
LIN {X 0,Y 175.074,Z 751.198,A -85,B 0,C 180,E1 -23579.037,E2 -23579.037} C_VEL
LIN {X 0,Y 176.665,Z 754.497,A -85,B 0,C 180,E1 -23581.746,E2 -23581.746} C_VEL
LIN {X 0,Y 179.06,Z 756.811,A -85,B 0,C 180,E1 -23584.644,E2 -23584.644} C_VEL
LIN {X 0,Y 181.398,Z 760.312,A -85,B 0,C 180,E1 -23587.105,E2 -23587.105} C_VEL
LIN {X 0,Y 182.452,Z 761.627,A -85,B 0,C 180,E1 -23588.082,E2 -23588.082} C_VEL
LIN {X 0,Y 185.119,Z 765.426,A -85,B 0,C 180,E1 -23590.339,E2 -23590.339} C_VEL
LIN {X 0,Y 188.977,Z 771.246,A -85,B 0,C 180,E1 -23593.208,E2 -23593.208} C_VEL
LIN {X 0,Y 193.125,Z 777.73,A -85,B 0,C 180,E1 -23595.849,E2 -23595.849} C_VEL
LIN {X 0,Y 198.111,Z 786.509,A -85,B 0,C 180,E1 -23598.689,E2 -23598.689} C_VEL
LIN {X 0,Y 201.692,Z 793.737,A -85,B 0,C 180,E1 -23600.561,E2 -23600.561} C_VEL
LIN {X 0,Y 200.04,Z 822.82,A -85,B 0,C 180,E1 -23601.833,E2 -23601.833} C_VEL
LIN {X 0,Y 198.546,Z 836.191,A -85,B 0,C 180,E1 -23602.797,E2 -23602.797} C_VEL
LIN {X 0,Y 196.286,Z 848.866,A -85,B 0,C 180,E1 -23604.082,E2 -23604.082} C_VEL
LIN {X 0,Y 193.134,Z 861.119,A -85,B 0,C 180,E1 -23605.741,E2 -23605.741} C_VEL
LIN {X 0,Y 189.577,Z 872.209,A -85,B 0,C 180,E1 -23607.718,E2 -23607.718} C_VEL
LIN {X 0,Y 185.611,Z 882.205,A -85,B 0,C 180,E1 -23609.994,E2 -23609.994} C_VEL
LIN {X 0,Y 181.376,Z 891.258,A -85,B 0,C 180,E1 -23612.634,E2 -23612.634} C_VEL
LIN {X 0,Y 177.163,Z 899.162,A -85,B 0,C 180,E1 -23615.594,E2 -23615.594} C_VEL
LIN {X 0,Y 173.274,Z 905.574,A -85,B 0,C 180,E1 -23618.674,E2 -23618.674} C_VEL
LIN {X 0,Y 169.883,Z 910.694,A -85,B 0,C 180,E1 -23621.876,E2 -23621.876} C_VEL
LIN {X 0,Y 166.152,Z 915.564,A -85,B 0,C 180,E1 -23625.979,E2 -23625.979} C_VEL
LIN {X 0,Y 163.373,Z 918.72,A -85,B 0,C 180,E1 -23629.819,E2 -23629.819} C_VEL
LIN {X 0,Y 161.861,Z 920.267,A -85,B 0,C 180,E1 -23632.569,E2 -23632.569} C_VEL
LIN {X 0,Y 160.183,Z 921.559,A -85,B 0,C 180,E1 -23636.474,E2 -23636.474} C_VEL
LIN {X 0,Y 158.958,Z 921.875,A -85,B 0,C 180,E1 -23640.904,E2 -23640.904} C_VEL
LIN {X 0,Y 158.514,Z 921.438,A -85,B 0,C 180,E1 -23643.686,E2 -23643.686} C_VEL
LIN {X 0,Y 158.48,Z 919.549,A -85,B 0,C 180,E1 -23648.636,E2 -23648.636} C_VEL
LIN {X 0,Y 159.28,Z 916.298,A -85,B 0,C 180,E1 -23653.337,E2 -23653.337} C_VEL
LIN {X 0,Y 160.599,Z 912.25,A -85,B 0,C 180,E1 -23657.365,E2 -23657.365} C_VEL
LIN {X 0,Y 162.392,Z 907.003,A -85,B 0,C 180,E1 -23661.293,E2 -23661.293} C_VEL
LIN {X 0,Y 164.729,Z 900.392,A -85,B 0,C 180,E1 -23665.109,E2 -23665.109} C_VEL
LIN {X 0,Y 167.027,Z 893.648,A -85,B 0,C 180,E1 -23668.195,E2 -23668.195} C_VEL
LIN {X 0,Y 169.705,Z 885.319,A -85,B 0,C 180,E1 -23671.266,E2 -23671.266} C_VEL
LIN {X 0,Y 172.543,Z 875.637,A -85,B 0,C 180,E1 -23674.091,E2 -23674.091} C_VEL
LIN {X 0,Y 175.359,Z 864.675,A -85,B 0,C 180,E1 -23676.62,E2 -23676.62} C_VEL
LIN {X 0,Y 177.896,Z 853.038,A -85,B 0,C 180,E1 -23678.693,E2 -23678.693} C_VEL
LIN {X 0,Y 180.01,Z 840.378,A -85,B 0,C 180,E1 -23680.406,E2 -23680.406} C_VEL
LIN {X 0,Y 181.532,Z 827.139,A -85,B 0,C 180,E1 -23681.712,E2 -23681.712} C_VEL
LIN {X 0,Y 182.367,Z 813.634,A -85,B 0,C 180,E1 -23682.584,E2 -23682.584} C_VEL
LIN {X 0,Y 183.58,Z 780.218,A -85,B 0,C 180,E1 -23684.002,E2 -23684.002} C_VEL
LIN {X 0,Y 177.025,Z 766.184,A -85,B 0,C 180,E1 -23686.175,E2 -23686.175} C_VEL
LIN {X 0,Y 168.694,Z 751.473,A -85,B 0,C 180,E1 -23689.093,E2 -23689.093} C_VEL
LIN {X 0,Y 162.426,Z 741.421,A -85,B 0,C 180,E1 -23691.491,E2 -23691.491} C_VEL
LIN {X 0,Y 159.454,Z 737.144,A -85,B 0,C 180,E1 -23692.688,E2 -23692.688} C_VEL
LIN {X 0,Y 157.667,Z 734.506,A -85,B 0,C 180,E1 -23693.447,E2 -23693.447} C_VEL
LIN {X 0,Y 157.323,Z 733.276,A -85,B 0,C 180,E1 -23693.885,E2 -23693.885} C_VEL
LIN {X 0,Y 157.301,Z 732.862,A -85,B 0,C 180,E1 -23695.12,E2 -23695.12} C_VEL
LIN {X 0,Y 157.236,Z 732.888,A -85,B 0,C 180,E1 -23699.454,E2 -23699.454} C_VEL
LIN {X 0,Y 157.267,Z 732.864,A -85,B 0,C 180,E1 -23702.434,E2 -23702.434} C_VEL
LIN {X 0,Y 157.265,Z 732.853,A -85,B 0,C 180,E1 -23706.447,E2 -23706.447} C_VEL
LIN {X 0,Y 157.217,Z 732.903,A -85,B 0,C 180,E1 -23712.113,E2 -23712.113} C_VEL
LIN {X 0,Y 157.302,Z 733.229,A -85,B 0,C 180,E1 -23713.628,E2 -23713.628} C_VEL
LIN {X 0,Y 157.641,Z 734.538,A -85,B 0,C 180,E1 -23713.966,E2 -23713.966} C_VEL
LIN {X 0,Y 168.11,Z 765.561,A -85,B 0,C 180,E1 -23717.137,E2 -23717.137} C_VEL
LIN {X 0,Y 165.811,Z 814.809,A -85,B 0,C 180,E1 -23720.465,E2 -23720.465} C_VEL
LIN {X 0,Y 164.947,Z 826.961,A -85,B 0,C 180,E1 -23721.648,E2 -23721.648} C_VEL
LIN {X 0,Y 164.024,Z 837.188,A -85,B 0,C 180,E1 -23722.947,E2 -23722.947} C_VEL
LIN {X 0,Y 163.102,Z 846.507,A -85,B 0,C 180,E1 -23724.402,E2 -23724.402} C_VEL
LIN {X 0,Y 162.109,Z 855.45,A -85,B 0,C 180,E1 -23726.07,E2 -23726.07} C_VEL
LIN {X 0,Y 160.913,Z 865.736,A -85,B 0,C 180,E1 -23728.391,E2 -23728.391} C_VEL
LIN {X 0,Y 159.814,Z 874.363,A -85,B 0,C 180,E1 -23730.709,E2 -23730.709} C_VEL
LIN {X 0,Y 158.883,Z 882.267,A -85,B 0,C 180,E1 -23733.198,E2 -23733.198} C_VEL
LIN {X 0,Y 158.24,Z 889.24,A -85,B 0,C 180,E1 -23735.743,E2 -23735.743} C_VEL
LIN {X 0,Y 157.606,Z 896.932,A -85,B 0,C 180,E1 -23739.099,E2 -23739.099} C_VEL
LIN {X 0,Y 157.336,Z 903.369,A -85,B 0,C 180,E1 -23742.451,E2 -23742.451} C_VEL
LIN {X 0,Y 157.426,Z 908.776,A -85,B 0,C 180,E1 -23745.786,E2 -23745.786} C_VEL
LIN {X 0,Y 158.142,Z 914.044,A -85,B 0,C 180,E1 -23749.76,E2 -23749.76} C_VEL
LIN {X 0,Y 159.434,Z 918.136,A -85,B 0,C 180,E1 -23753.673,E2 -23753.673} C_VEL
LIN {X 0,Y 161.749,Z 921.542,A -85,B 0,C 180,E1 -23758.03,E2 -23758.03} C_VEL
LIN {X 0,Y 163.051,Z 922.8,A -85,B 0,C 180,E1 -23760,E2 -23760} C_VEL
LIN {X 0,Y 165.012,Z 923.871,A -85,B 0,C 180,E1 -23762.441,E2 -23762.441} C_VEL
LIN {X 0,Y 169.673,Z 924.809,A -85,B 0,C 180,E1 -23767.138,E2 -23767.138} C_VEL
LIN {X 0,Y 175.356,Z 924.106,A -85,B 0,C 180,E1 -23771.56,E2 -23771.56} C_VEL
LIN {X 0,Y 178.605,Z 923.13,A -85,B 0,C 180,E1 -23773.656,E2 -23773.656} C_VEL
LIN {X 0,Y 185.736,Z 919.966,A -85,B 0,C 180,E1 -23777.62,E2 -23777.62} C_VEL
LIN {X 0,Y 191.621,Z 916.385,A -85,B 0,C 180,E1 -23780.391,E2 -23780.391} C_VEL
LIN {X 0,Y 197.875,Z 911.726,A -85,B 0,C 180,E1 -23782.997,E2 -23782.997} C_VEL
LIN {X 0,Y 203.429,Z 906.928,A -85,B 0,C 180,E1 -23785.037,E2 -23785.037} C_VEL
LIN {X 0,Y 210.356,Z 899.845,A -85,B 0,C 180,E1 -23787.347,E2 -23787.347} C_VEL
LIN {X 0,Y 216.328,Z 892.759,A -85,B 0,C 180,E1 -23789.164,E2 -23789.164} C_VEL
LIN {X 0,Y 222.201,Z 884.697,A -85,B 0,C 180,E1 -23790.805,E2 -23790.805} C_VEL
LIN {X 0,Y 226.955,Z 877.201,A -85,B 0,C 180,E1 -23792.064,E2 -23792.064} C_VEL
LIN {X 0,Y 231.957,Z 867.938,A -85,B 0,C 180,E1 -23793.309,E2 -23793.309} C_VEL
LIN {X 0,Y 236.366,Z 858.335,A -85,B 0,C 180,E1 -23794.398,E2 -23794.398} C_VEL
LIN {X 0,Y 239.736,Z 849.409,A -85,B 0,C 180,E1 -23795.216,E2 -23795.216} C_VEL
LIN {X 0,Y 242.856,Z 839.035,A -85,B 0,C 180,E1 -23796.006,E2 -23796.006} C_VEL
